LIN {X 0,Y 359.828,Z 337.187,A -85,B 0,C 180,E1 -13571.495,E2 -13571.495} C_VEL
LIN {X 0,Y 358.467,Z 346.595,A -85,B 0,C 180,E1 -13572.897,E2 -13572.897} C_VEL
LIN {X 0,Y 356.952,Z 356.826,A -85,B 0,C 180,E1 -13574.744,E2 -13574.744} C_VEL
LIN {X 0,Y 355.949,Z 365.054,A -85,B 0,C 180,E1 -13576.585,E2 -13576.585} C_VEL
LIN {X 0,Y 354.906,Z 372.31,A -85,B 0,C 180,E1 -13578.579,E2 -13578.579} C_VEL
LIN {X 0,Y 354.13,Z 378.825,A -85,B 0,C 180,E1 -13580.865,E2 -13580.865} C_VEL
LIN {X 0,Y 353.677,Z 383.707,A -85,B 0,C 180,E1 -13583.153,E2 -13583.153} C_VEL
LIN {X 0,Y 353.389,Z 387.105,A -85,B 0,C 180,E1 -13585.437,E2 -13585.437} C_VEL
LIN {X 0,Y 353.199,Z 389.123,A -85,B 0,C 180,E1 -13587.719,E2 -13587.719} C_VEL
LIN {X 0,Y 353.194,Z 389.814,A -85,B 0,C 180,E1 -13590,E2 -13590} C_VEL
LIN {X 0,Y 353.198,Z 389.189,A -85,B 0,C 180,E1 -13592.281,E2 -13592.281} C_VEL
LIN {X 0,Y 353.386,Z 387.229,A -85,B 0,C 180,E1 -13594.563,E2 -13594.563} C_VEL
LIN {X 0,Y 353.675,Z 383.892,A -85,B 0,C 180,E1 -13596.848,E2 -13596.848} C_VEL
LIN {X 0,Y 354.107,Z 379.078,A -85,B 0,C 180,E1 -13599.136,E2 -13599.136} C_VEL
LIN {X 0,Y 354.636,Z 374.431,A -85,B 0,C 180,E1 -13600.852,E2 -13600.852} C_VEL
LIN {X 0,Y 355.584,Z 367.668,A -85,B 0,C 180,E1 -13602.847,E2 -13602.847} C_VEL
LIN {X 0,Y 356.525,Z 360.612,A -85,B 0,C 180,E1 -13604.557,E2 -13604.557} C_VEL
LIN {X 0,Y 357.678,Z 352.114,A -85,B 0,C 180,E1 -13606.26,E2 -13606.26} C_VEL
LIN {X 0,Y 359.22,Z 341.807,A -85,B 0,C 180,E1 -13607.948,E2 -13607.948} C_VEL
LIN {X 0,Y 360.78,Z 330.276,A -85,B 0,C 180,E1 -13609.487,E2 -13609.487} C_VEL
LIN {X 0,Y 362.233,Z 318.754,A -85,B 0,C 180,E1 -13610.738,E2 -13610.738} C_VEL
LIN {X 0,Y 363.624,Z 305.23,A -85,B 0,C 180,E1 -13611.916,E2 -13611.916} C_VEL
LIN {X 0,Y 364.064,Z 298.662,A -85,B 0,C 180,E1 -13612.398,E2 -13612.398} C_VEL
LIN {X 0,Y 361.429,Z 285.746,A -85,B 0,C 180,E1 -13613.406,E2 -13613.406} C_VEL
LIN {X 0,Y 357.948,Z 272.835,A -85,B 0,C 180,E1 -13614.268,E2 -13614.268} C_VEL
LIN {X 0,Y 354.079,Z 260.487,A -85,B 0,C 180,E1 -13614.972,E2 -13614.972} C_VEL
LIN {X 0,Y 354.298,Z 256.381,A -85,B 0,C 180,E1 -13618.43,E2 -13618.43} C_VEL
LIN {X 0,Y 354.484,Z 253.656,A -85,B 0,C 180,E1 -13620.771,E2 -13620.771} C_VEL
LIN {X 0,Y 353.931,Z 252.674,A -85,B 0,C 180,E1 -13621.708,E2 -13621.708} C_VEL
LIN {X 0,Y 351.187,Z 251.333,A -85,B 0,C 180,E1 -13623.242,E2 -13623.242} C_VEL
LIN {X 0,Y 348.857,Z 250.304,A -85,B 0,C 180,E1 -13624.486,E2 -13624.486} C_VEL
LIN {X 0,Y 347.923,Z 249.415,A -85,B 0,C 180,E1 -13625.443,E2 -13625.443} C_VEL
LIN {X 0,Y 347.886,Z 249.081,A -85,B 0,C 180,E1 -13625.766,E2 -13625.766} C_VEL
LIN {X 0,Y 347.949,Z 246.009,A -85,B 0,C 180,E1 -13628.767,E2 -13628.767} C_VEL
LIN {X 0,Y 347.764,Z 243.044,A -85,B 0,C 180,E1 -13631.829,E2 -13631.829} C_VEL
LIN {X 0,Y 347.707,Z 242.802,A -85,B 0,C 180,E1 -13635.027,E2 -13635.027} C_VEL
LIN {X 0,Y 347.743,Z 242.796,A -85,B 0,C 180,E1 -13638.399,E2 -13638.399} C_VEL
LIN {X 0,Y 347.759,Z 242.794,A -85,B 0,C 180,E1 -13642.679,E2 -13642.679} C_VEL
LIN {X 0,Y 347.751,Z 242.795,A -85,B 0,C 180,E1 -13645.956,E2 -13645.956} C_VEL
LIN {X 0,Y 347.752,Z 242.794,A -85,B 0,C 180,E1 -13649.652,E2 -13649.652} C_VEL
LIN {X 0,Y 347.833,Z 242.783,A -85,B 0,C 180,E1 -13653.608,E2 -13653.608} C_VEL
LIN {X 0,Y 347.788,Z 242.789,A -85,B 0,C 180,E1 -13656.162,E2 -13656.162} C_VEL
LIN {X 0,Y 347.809,Z 242.783,A -85,B 0,C 180,E1 -13659.909,E2 -13659.909} C_VEL
LIN {X 0,Y 347.869,Z 242.779,A -85,B 0,C 180,E1 -13662.359,E2 -13662.359} C_VEL
LIN {X 0,Y 347.9,Z 242.773,A -85,B 0,C 180,E1 -13665.971,E2 -13665.971} C_VEL
LIN {X 0,Y 347.899,Z 242.772,A -85,B 0,C 180,E1 -13669.525,E2 -13669.525} C_VEL
LIN {X 0,Y 348.081,Z 242.751,A -85,B 0,C 180,E1 -13673.042,E2 -13673.042} C_VEL
LIN {X 0,Y 348.205,Z 242.734,A -85,B 0,C 180,E1 -13677.686,E2 -13677.686} C_VEL
LIN {X 0,Y 348.151,Z 242.743,A -85,B 0,C 180,E1 -13681.157,E2 -13681.157} C_VEL
LIN {X 0,Y 348.208,Z 242.733,A -85,B 0,C 180,E1 -13682.313,E2 -13682.313} C_VEL
LIN {X 0,Y 348.058,Z 242.753,A -85,B 0,C 180,E1 -13686.959,E2 -13686.959} C_VEL
LIN {X 0,Y 347.899,Z 242.774,A -85,B 0,C 180,E1 -13690.475,E2 -13690.475} C_VEL
LIN {X 0,Y 347.901,Z 242.775,A -85,B 0,C 180,E1 -13694.15,E2 -13694.15} C_VEL
LIN {X 0,Y 347.832,Z 242.783,A -85,B 0,C 180,E1 -13698.259,E2 -13698.259} C_VEL
LIN {X 0,Y 347.77,Z 242.791,A -85,B 0,C 180,E1 -13701.626,E2 -13701.626} C_VEL
LIN {X 0,Y 347.77,Z 242.787,A -85,B 0,C 180,E1 -13705.112,E2 -13705.112} C_VEL
LIN {X 0,Y 347.747,Z 242.795,A -85,B 0,C 180,E1 -13709.015,E2 -13709.015} C_VEL
LIN {X 0,Y 347.74,Z 242.793,A -85,B 0,C 180,E1 -13711.914,E2 -13711.914} C_VEL
LIN {X 0,Y 347.79,Z 242.793,A -85,B 0,C 180,E1 -13715.875,E2 -13715.875} C_VEL
LIN {X 0,Y 347.754,Z 242.795,A -85,B 0,C 180,E1 -13718.792,E2 -13718.792} C_VEL
LIN {X 0,Y 347.773,Z 242.876,A -85,B 0,C 180,E1 -13722.962,E2 -13722.962} C_VEL
LIN {X 0,Y 348.43,Z 246.978,A -85,B 0,C 180,E1 -13726.564,E2 -13726.564} C_VEL
LIN {X 0,Y 348.931,Z 251.04,A -85,B 0,C 180,E1 -13729.869,E2 -13729.869} C_VEL
LIN {X 0,Y 348.958,Z 253.507,A -85,B 0,C 180,E1 -13731.763,E2 -13731.763} C_VEL
LIN {X 0,Y 348.65,Z 256.872,A -85,B 0,C 180,E1 -13734.227,E2 -13734.227} C_VEL
LIN {X 0,Y 348.101,Z 262.637,A -85,B 0,C 180,E1 -13738.336,E2 -13738.336} C_VEL
LIN {X 0,Y 347.747,Z 266.494,A -85,B 0,C 180,E1 -13740.984,E2 -13740.984} C_VEL
LIN {X 0,Y 347.238,Z 271.759,A -85,B 0,C 180,E1 -13744.526,E2 -13744.526} C_VEL
LIN {X 0,Y 351.846,Z 288.484,A -85,B 0,C 180,E1 -13745.474,E2 -13745.474} C_VEL
LIN {X 0,Y 354.51,Z 300.834,A -85,B 0,C 180,E1 -13746.312,E2 -13746.312} C_VEL
LIN {X 0,Y 356.336,Z 312.535,A -85,B 0,C 180,E1 -13747.231,E2 -13747.231} C_VEL
LIN {X 0,Y 356.681,Z 316.48,A -85,B 0,C 180,E1 -13747.559,E2 -13747.559} C_VEL
LIN {X 0,Y 355.212,Z 330.023,A -85,B 0,C 180,E1 -13748.725,E2 -13748.725} C_VEL
LIN {X 0,Y 353.479,Z 342.684,A -85,B 0,C 180,E1 -13750.093,E2 -13750.093} C_VEL
LIN {X 0,Y 351.824,Z 354.335,A -85,B 0,C 180,E1 -13751.662,E2 -13751.662} C_VEL
LIN {X 0,Y 350.3,Z 364.758,A -85,B 0,C 180,E1 -13753.387,E2 -13753.387} C_VEL
LIN {X 0,Y 349.048,Z 374.137,A -85,B 0,C 180,E1 -13755.304,E2 -13755.304} C_VEL
LIN {X 0,Y 348.046,Z 381.599,A -85,B 0,C 180,E1 -13757.166,E2 -13757.166} C_VEL
LIN {X 0,Y 347.207,Z 387.367,A -85,B 0,C 180,E1 -13758.913,E2 -13758.913} C_VEL
LIN {X 0,Y 346.726,Z 392.095,A -85,B 0,C 180,E1 -13760.668,E2 -13760.668} C_VEL
LIN {X 0,Y 346.337,Z 396.996,A -85,B 0,C 180,E1 -13763.007,E2 -13763.007} C_VEL
LIN {X 0,Y 346.143,Z 400.404,A -85,B 0,C 180,E1 -13765.341,E2 -13765.341} C_VEL
LIN {X 0,Y 346.053,Z 402.419,A -85,B 0,C 180,E1 -13767.672,E2 -13767.672} C_VEL
LIN {X 0,Y 346.092,Z 403.086,A -85,B 0,C 180,E1 -13770,E2 -13770} C_VEL
LIN {X 0,Y 346.053,Z 402.413,A -85,B 0,C 180,E1 -13772.328,E2 -13772.328} C_VEL
LIN {X 0,Y 346.14,Z 400.393,A -85,B 0,C 180,E1 -13774.658,E2 -13774.658} C_VEL
LIN {X 0,Y 346.337,Z 396.976,A -85,B 0,C 180,E1 -13776.993,E2 -13776.993} C_VEL
LIN {X 0,Y 346.716,Z 392.062,A -85,B 0,C 180,E1 -13779.332,E2 -13779.332} C_VEL
LIN {X 0,Y 347.431,Z 385.508,A -85,B 0,C 180,E1 -13781.671,E2 -13781.671} C_VEL
LIN {X 0,Y 348.302,Z 379.34,A -85,B 0,C 180,E1 -13783.417,E2 -13783.417} C_VEL
LIN {X 0,Y 349.285,Z 371.939,A -85,B 0,C 180,E1 -13785.163,E2 -13785.163} C_VEL
LIN {X 0,Y 350.526,Z 363.049,A -85,B 0,C 180,E1 -13786.901,E2 -13786.901} C_VEL
LIN {X 0,Y 352.091,Z 352.286,A -85,B 0,C 180,E1 -13788.625,E2 -13788.625} C_VEL
LIN {X 0,Y 353.64,Z 341.395,A -85,B 0,C 180,E1 -13790.048,E2 -13790.048} C_VEL
LIN {X 0,Y 355.281,Z 329.679,A -85,B 0,C 180,E1 -13791.293,E2 -13791.293} C_VEL
LIN {X 0,Y 356.654,Z 316.345,A -85,B 0,C 180,E1 -13792.439,E2 -13792.439} C_VEL
LIN {X 0,Y 355.141,Z 304.648,A -85,B 0,C 180,E1 -13793.392,E2 -13793.392} C_VEL
LIN {X 0,Y 352.32,Z 290.353,A -85,B 0,C 180,E1 -13794.393,E2 -13794.393} C_VEL
LIN {X 0,Y 348.517,Z 276.599,A -85,B 0,C 180,E1 -13795.205,E2 -13795.205} C_VEL
LIN {X 0,Y 347.245,Z 271.771,A -85,B 0,C 180,E1 -13795.448,E2 -13795.448} C_VEL
LIN {X 0,Y 347.745,Z 266.467,A -85,B 0,C 180,E1 -13799.015,E2 -13799.015} C_VEL
LIN {X 0,Y 348.262,Z 260.693,A -85,B 0,C 180,E1 -13803.016,E2 -13803.016} C_VEL
LIN {X 0,Y 348.722,Z 256.134,A -85,B 0,C 180,E1 -13806.279,E2 -13806.279} C_VEL
LIN {X 0,Y 348.962,Z 252.942,A -85,B 0,C 180,E1 -13808.633,E2 -13808.633} C_VEL
LIN {X 0,Y 348.927,Z 250.987,A -85,B 0,C 180,E1 -13810.131,E2 -13810.131} C_VEL
LIN {X 0,Y 348.416,Z 246.945,A -85,B 0,C 180,E1 -13813.434,E2 -13813.434} C_VEL
LIN {X 0,Y 347.845,Z 243.239,A -85,B 0,C 180,E1 -13816.666,E2 -13816.666} C_VEL
LIN {X 0,Y 347.755,Z 242.797,A -85,B 0,C 180,E1 -13817.226,E2 -13817.226} C_VEL
LIN {X 0,Y 347.752,Z 242.796,A -85,B 0,C 180,E1 -13821.207,E2 -13821.207} C_VEL
LIN {X 0,Y 347.789,Z 242.792,A -85,B 0,C 180,E1 -13824.125,E2 -13824.125} C_VEL
LIN {X 0,Y 347.739,Z 242.796,A -85,B 0,C 180,E1 -13828.086,E2 -13828.086} C_VEL
LIN {X 0,Y 347.747,Z 242.795,A -85,B 0,C 180,E1 -13830.985,E2 -13830.985} C_VEL
LIN {X 0,Y 347.751,Z 242.793,A -85,B 0,C 180,E1 -13833.601,E2 -13833.601} C_VEL
LIN {X 0,Y 347.77,Z 242.791,A -85,B 0,C 180,E1 -13836.161,E2 -13836.161} C_VEL
LIN {X 0,Y 347.807,Z 242.786,A -85,B 0,C 180,E1 -13839.909,E2 -13839.909} C_VEL
LIN {X 0,Y 347.834,Z 242.783,A -85,B 0,C 180,E1 -13843.568,E2 -13843.568} C_VEL
LIN {X 0,Y 347.891,Z 242.777,A -85,B 0,C 180,E1 -13847.161,E2 -13847.161} C_VEL
LIN {X 0,Y 347.936,Z 242.77,A -85,B 0,C 180,E1 -13850.701,E2 -13850.701} C_VEL
LIN {X 0,Y 348.045,Z 242.755,A -85,B 0,C 180,E1 -13854.205,E2 -13854.205} C_VEL
LIN {X 0,Y 348.207,Z 242.735,A -85,B 0,C 180,E1 -13857.687,E2 -13857.687} C_VEL
LIN {X 0,Y 348.284,Z 242.728,A -85,B 0,C 180,E1 -13860,E2 -13860} C_VEL
LIN {X 0,Y 348.203,Z 242.735,A -85,B 0,C 180,E1 -13862.314,E2 -13862.314} C_VEL
LIN {X 0,Y 348.092,Z 242.75,A -85,B 0,C 180,E1 -13866.958,E2 -13866.958} C_VEL
LIN {X 0,Y 347.93,Z 242.77,A -85,B 0,C 180,E1 -13870.474,E2 -13870.474} C_VEL
LIN {X 0,Y 347.9,Z 242.773,A -85,B 0,C 180,E1 -13874.15,E2 -13874.15} C_VEL
LIN {X 0,Y 347.893,Z 242.775,A -85,B 0,C 180,E1 -13878.291,E2 -13878.291} C_VEL
LIN {X 0,Y 347.769,Z 242.789,A -85,B 0,C 180,E1 -13881.626,E2 -13881.626} C_VEL
LIN {X 0,Y 347.813,Z 242.784,A -85,B 0,C 180,E1 -13885.109,E2 -13885.109} C_VEL
LIN {X 0,Y 347.81,Z 242.786,A -85,B 0,C 180,E1 -13887.694,E2 -13887.694} C_VEL
LIN {X 0,Y 347.751,Z 242.793,A -85,B 0,C 180,E1 -13890.348,E2 -13890.348} C_VEL
LIN {X 0,Y 347.749,Z 242.794,A -85,B 0,C 180,E1 -13894.044,E2 -13894.044} C_VEL
LIN {X 0,Y 347.758,Z 242.794,A -85,B 0,C 180,E1 -13897.322,E2 -13897.322} C_VEL
LIN {X 0,Y 347.742,Z 242.796,A -85,B 0,C 180,E1 -13901.601,E2 -13901.601} C_VEL
LIN {X 0,Y 347.706,Z 242.8,A -85,B 0,C 180,E1 -13905.027,E2 -13905.027} C_VEL
LIN {X 0,Y 347.763,Z 242.921,A -85,B 0,C 180,E1 -13908.172,E2 -13908.172} C_VEL
LIN {X 0,Y 347.964,Z 245.902,A -85,B 0,C 180,E1 -13911.235,E2 -13911.235} C_VEL
LIN {X 0,Y 347.897,Z 248.859,A -85,B 0,C 180,E1 -13914.138,E2 -13914.138} C_VEL
LIN {X 0,Y 347.633,Z 251.861,A -85,B 0,C 180,E1 -13916.917,E2 -13916.917} C_VEL
LIN {X 0,Y 347.313,Z 255.844,A -85,B 0,C 180,E1 -13920.473,E2 -13920.473} C_VEL
LIN {X 0,Y 347.05,Z 260.626,A -85,B 0,C 180,E1 -13924.592,E2 -13924.592} C_VEL
LIN {X 0,Y 352.324,Z 277.531,A -85,B 0,C 180,E1 -13925.624,E2 -13925.624} C_VEL
LIN {X 0,Y 355.52,Z 290.249,A -85,B 0,C 180,E1 -13926.55,E2 -13926.55} C_VEL
LIN {X 0,Y 357.453,Z 300.982,A -85,B 0,C 180,E1 -13927.439,E2 -13927.439} C_VEL
LIN {X 0,Y 356.211,Z 313.402,A -85,B 0,C 180,E1 -13928.44,E2 -13928.44} C_VEL
LIN {X 0,Y 354.679,Z 325.974,A -85,B 0,C 180,E1 -13929.71,E2 -13929.71} C_VEL
LIN {X 0,Y 353.104,Z 337.325,A -85,B 0,C 180,E1 -13931.129,E2 -13931.129} C_VEL
LIN {X 0,Y 351.68,Z 346.733,A -85,B 0,C 180,E1 -13932.557,E2 -13932.557} C_VEL
LIN {X 0,Y 350.18,Z 356.452,A -85,B 0,C 180,E1 -13934.334,E2 -13934.334} C_VEL
LIN {X 0,Y 349.021,Z 365.191,A -85,B 0,C 180,E1 -13936.314,E2 -13936.314} C_VEL
LIN {X 0,Y 347.905,Z 372.448,A -85,B 0,C 180,E1 -13938.346,E2 -13938.346} C_VEL
LIN {X 0,Y 347.111,Z 378.961,A -85,B 0,C 180,E1 -13940.678,E2 -13940.678} C_VEL
LIN {X 0,Y 346.613,Z 383.843,A -85,B 0,C 180,E1 -13943.012,E2 -13943.012} C_VEL
LIN {X 0,Y 346.308,Z 387.24,A -85,B 0,C 180,E1 -13945.344,E2 -13945.344} C_VEL
LIN {X 0,Y 346.11,Z 389.258,A -85,B 0,C 180,E1 -13947.673,E2 -13947.673} C_VEL
LIN {X 0,Y 346.095,Z 389.949,A -85,B 0,C 180,E1 -13950,E2 -13950} C_VEL
LIN {X 0,Y 346.109,Z 389.323,A -85,B 0,C 180,E1 -13952.328,E2 -13952.328} C_VEL
LIN {X 0,Y 346.304,Z 387.363,A -85,B 0,C 180,E1 -13954.656,E2 -13954.656} C_VEL
LIN {X 0,Y 346.612,Z 384.026,A -85,B 0,C 180,E1 -13956.988,E2 -13956.988} C_VEL
LIN {X 0,Y 347.093,Z 379.212,A -85,B 0,C 180,E1 -13959.322,E2 -13959.322} C_VEL
LIN {X 0,Y 347.844,Z 372.765,A -85,B 0,C 180,E1 -13961.657,E2 -13961.657} C_VEL
LIN {X 0,Y 348.99,Z 365.579,A -85,B 0,C 180,E1 -13963.687,E2 -13963.687} C_VEL
LIN {X 0,Y 350.126,Z 356.973,A -85,B 0,C 180,E1 -13965.663,E2 -13965.663} C_VEL
LIN {X 0,Y 351.645,Z 347.35,A -85,B 0,C 180,E1 -13967.445,E2 -13967.445} C_VEL
LIN {X 0,Y 353.161,Z 337.001,A -85,B 0,C 180,E1 -13969.018,E2 -13969.018} C_VEL
LIN {X 0,Y 354.73,Z 325.578,A -85,B 0,C 180,E1 -13970.438,E2 -13970.438} C_VEL
LIN {X 0,Y 356.287,Z 312.912,A -85,B 0,C 180,E1 -13971.707,E2 -13971.707} C_VEL
LIN {X 0,Y 357.481,Z 300.595,A -85,B 0,C 180,E1 -13972.695,E2 -13972.695} C_VEL
LIN {X 0,Y 354.933,Z 287.672,A -85,B 0,C 180,E1 -13973.753,E2 -13973.753} C_VEL
LIN {X 0,Y 351.396,Z 274.214,A -85,B 0,C 180,E1 -13974.696,E2 -13974.696} C_VEL
LIN {X 0,Y 347.12,Z 261.12,A -85,B 0,C 180,E1 -13975.472,E2 -13975.472} C_VEL
LIN {X 0,Y 347.057,Z 260.623,A -85,B 0,C 180,E1 -13975.52,E2 -13975.52} C_VEL
LIN {X 0,Y 347.342,Z 255.956,A -85,B 0,C 180,E1 -13979.536,E2 -13979.536} C_VEL
LIN {X 0,Y 347.634,Z 251.985,A -85,B 0,C 180,E1 -13983.083,E2 -13983.083} C_VEL
LIN {X 0,Y 347.886,Z 249.081,A -85,B 0,C 180,E1 -13985.766,E2 -13985.766} C_VEL
LIN {X 0,Y 347.327,Z 248.172,A -85,B 0,C 180,E1 -13986.72,E2 -13986.72} C_VEL
LIN {X 0,Y 344.517,Z 247.005,A -85,B 0,C 180,E1 -13988.281,E2 -13988.281} C_VEL
LIN {X 0,Y 342.041,Z 246.131,A -85,B 0,C 180,E1 -13989.546,E2 -13989.546} C_VEL
LIN {X 0,Y 340.928,Z 245.355,A -85,B 0,C 180,E1 -13990.523,E2 -13990.523} C_VEL
LIN {X 0,Y 340.815,Z 245.056,A -85,B 0,C 180,E1 -13990.853,E2 -13990.853} C_VEL
LIN {X 0,Y 340.727,Z 243.941,A -85,B 0,C 180,E1 -13992.05,E2 -13992.05} C_VEL
LIN {X 0,Y 340.643,Z 243.682,A -85,B 0,C 180,E1 -13994.546,E2 -13994.546} C_VEL
LIN {X 0,Y 340.695,Z 243.674,A -85,B 0,C 180,E1 -13997.956,E2 -13997.956} C_VEL
LIN {X 0,Y 340.721,Z 243.668,A -85,B 0,C 180,E1 -14001.771,E2 -14001.771} C_VEL
LIN {X 0,Y 340.725,Z 243.668,A -85,B 0,C 180,E1 -14005.595,E2 -14005.595} C_VEL
LIN {X 0,Y 340.7,Z 243.672,A -85,B 0,C 180,E1 -14008.955,E2 -14008.955} C_VEL
LIN {X 0,Y 340.806,Z 243.658,A -85,B 0,C 180,E1 -14013.02,E2 -14013.02} C_VEL
LIN {X 0,Y 340.757,Z 243.661,A -85,B 0,C 180,E1 -14015.638,E2 -14015.638} C_VEL
LIN {X 0,Y 340.737,Z 243.665,A -85,B 0,C 180,E1 -14019.473,E2 -14019.473} C_VEL
LIN {X 0,Y 340.861,Z 243.652,A -85,B 0,C 180,E1 -14021.984,E2 -14021.984} C_VEL
LIN {X 0,Y 340.872,Z 243.65,A -85,B 0,C 180,E1 -14025.705,E2 -14025.705} C_VEL
LIN {X 0,Y 340.851,Z 243.65,A -85,B 0,C 180,E1 -14029.305,E2 -14029.305} C_VEL
LIN {X 0,Y 341.048,Z 243.627,A -85,B 0,C 180,E1 -14032.898,E2 -14032.898} C_VEL
LIN {X 0,Y 341.167,Z 243.611,A -85,B 0,C 180,E1 -14037.639,E2 -14037.639} C_VEL
LIN {X 0,Y 341.12,Z 243.619,A -85,B 0,C 180,E1 -14041.18,E2 -14041.18} C_VEL
LIN {X 0,Y 341.17,Z 243.61,A -85,B 0,C 180,E1 -14042.361,E2 -14042.361} C_VEL
LIN {X 0,Y 341.005,Z 243.631,A -85,B 0,C 180,E1 -14047.103,E2 -14047.103} C_VEL
LIN {X 0,Y 340.85,Z 243.652,A -85,B 0,C 180,E1 -14050.694,E2 -14050.694} C_VEL
LIN {X 0,Y 340.866,Z 243.652,A -85,B 0,C 180,E1 -14054.325,E2 -14054.325} C_VEL
LIN {X 0,Y 340.789,Z 243.66,A -85,B 0,C 180,E1 -14058.441,E2 -14058.441} C_VEL
LIN {X 0,Y 340.72,Z 243.669,A -85,B 0,C 180,E1 -14061.841,E2 -14061.841} C_VEL
LIN {X 0,Y 340.721,Z 243.664,A -85,B 0,C 180,E1 -14065.668,E2 -14065.668} C_VEL
LIN {X 0,Y 340.709,Z 243.671,A -85,B 0,C 180,E1 -14069.674,E2 -14069.674} C_VEL
LIN {X 0,Y 340.688,Z 243.675,A -85,B 0,C 180,E1 -14072.436,E2 -14072.436} C_VEL
LIN {X 0,Y 340.72,Z 243.672,A -85,B 0,C 180,E1 -14075.279,E2 -14075.279} C_VEL
LIN {X 0,Y 340.711,Z 243.673,A -85,B 0,C 180,E1 -14078.386,E2 -14078.386} C_VEL
LIN {X 0,Y 340.716,Z 243.722,A -85,B 0,C 180,E1 -14082.54,E2 -14082.54} C_VEL
LIN {X 0,Y 341.357,Z 247.68,A -85,B 0,C 180,E1 -14086.104,E2 -14086.104} C_VEL
LIN {X 0,Y 341.882,Z 251.744,A -85,B 0,C 180,E1 -14089.517,E2 -14089.517} C_VEL
LIN {X 0,Y 341.924,Z 254.813,A -85,B 0,C 180,E1 -14091.929,E2 -14091.929} C_VEL
LIN {X 0,Y 341.424,Z 259.506,A -85,B 0,C 180,E1 -14095.424,E2 -14095.424} C_VEL
LIN {X 0,Y 340.944,Z 264.434,A -85,B 0,C 180,E1 -14098.98,E2 -14098.98} C_VEL
LIN {X 0,Y 340.564,Z 268.275,A -85,B 0,C 180,E1 -14101.664,E2 -14101.664} C_VEL
LIN {X 0,Y 340.268,Z 271.798,A -85,B 0,C 180,E1 -14103.994,E2 -14103.994} C_VEL
LIN {X 0,Y 344.24,Z 285.702,A -85,B 0,C 180,E1 -14104.779,E2 -14104.779} C_VEL
LIN {X 0,Y 347.179,Z 298.328,A -85,B 0,C 180,E1 -14105.636,E2 -14105.636} C_VEL
LIN {X 0,Y 349.36,Z 311.042,A -85,B 0,C 180,E1 -14106.643,E2 -14106.643} C_VEL
LIN {X 0,Y 349.925,Z 318.302,A -85,B 0,C 180,E1 -14107.273,E2 -14107.273} C_VEL
LIN {X 0,Y 348.524,Z 330.344,A -85,B 0,C 180,E1 -14108.345,E2 -14108.345} C_VEL
LIN {X 0,Y 346.808,Z 342.553,A -85,B 0,C 180,E1 -14109.694,E2 -14109.694} C_VEL
LIN {X 0,Y 345.336,Z 352.247,A -85,B 0,C 180,E1 -14110.997,E2 -14110.997} C_VEL
LIN {X 0,Y 343.71,Z 362.992,A -85,B 0,C 180,E1 -14112.753,E2 -14112.753} C_VEL
LIN {X 0,Y 342.398,Z 371.868,A -85,B 0,C 180,E1 -14114.524,E2 -14114.524} C_VEL
LIN {X 0,Y 341.232,Z 380.377,A -85,B 0,C 180,E1 -14116.602,E2 -14116.602} C_VEL
LIN {X 0,Y 340.2,Z 387.233,A -85,B 0,C 180,E1 -14118.682,E2 -14118.682} C_VEL
LIN {X 0,Y 339.687,Z 391.961,A -85,B 0,C 180,E1 -14120.473,E2 -14120.473} C_VEL
LIN {X 0,Y 339.26,Z 396.862,A -85,B 0,C 180,E1 -14122.86,E2 -14122.86} C_VEL
LIN {X 0,Y 339.047,Z 400.27,A -85,B 0,C 180,E1 -14125.244,E2 -14125.244} C_VEL
LIN {X 0,Y 338.969,Z 402.285,A -85,B 0,C 180,E1 -14127.623,E2 -14127.623} C_VEL
LIN {X 0,Y 338.994,Z 402.951,A -85,B 0,C 180,E1 -14130,E2 -14130} C_VEL
LIN {X 0,Y 338.969,Z 402.278,A -85,B 0,C 180,E1 -14132.376,E2 -14132.376} C_VEL
LIN {X 0,Y 339.045,Z 400.257,A -85,B 0,C 180,E1 -14134.756,E2 -14134.756} C_VEL
LIN {X 0,Y 339.26,Z 396.84,A -85,B 0,C 180,E1 -14137.14,E2 -14137.14} C_VEL
LIN {X 0,Y 339.68,Z 391.926,A -85,B 0,C 180,E1 -14139.527,E2 -14139.527} C_VEL
LIN {X 0,Y 340.455,Z 385.371,A -85,B 0,C 180,E1 -14141.913,E2 -14141.913} C_VEL
LIN {X 0,Y 341.484,Z 378.081,A -85,B 0,C 180,E1 -14143.994,E2 -14143.994} C_VEL
LIN {X 0,Y 342.56,Z 370.441,A -85,B 0,C 180,E1 -14145.774,E2 -14145.774} C_VEL
LIN {X 0,Y 343.957,Z 361.279,A -85,B 0,C 180,E1 -14147.541,E2 -14147.541} C_VEL
LIN {X 0,Y 345.607,Z 350.169,A -85,B 0,C 180,E1 -14149.296,E2 -14149.296} C_VEL
LIN {X 0,Y 347.36,Z 338.831,A -85,B 0,C 180,E1 -14150.736,E2 -14150.736} C_VEL
LIN {X 0,Y 348.942,Z 327.034,A -85,B 0,C 180,E1 -14151.959,E2 -14151.959} C_VEL
LIN {X 0,Y 349.918,Z 316.488,A -85,B 0,C 180,E1 -14152.87,E2 -14152.87} C_VEL
LIN {X 0,Y 348.294,Z 304.5,A -85,B 0,C 180,E1 -14153.88,E2 -14153.88} C_VEL
LIN {X 0,Y 345.498,Z 290.644,A -85,B 0,C 180,E1 -14154.885,E2 -14154.885} C_VEL
LIN {X 0,Y 341.361,Z 275.824,A -85,B 0,C 180,E1 -14155.789,E2 -14155.789} C_VEL
LIN {X 0,Y 340.257,Z 271.653,A -85,B 0,C 180,E1 -14156.007,E2 -14156.007} C_VEL
LIN {X 0,Y 340.837,Z 265.842,A -85,B 0,C 180,E1 -14159.999,E2 -14159.999} C_VEL
LIN {X 0,Y 341.315,Z 260.561,A -85,B 0,C 180,E1 -14163.777,E2 -14163.777} C_VEL
LIN {X 0,Y 341.746,Z 256.635,A -85,B 0,C 180,E1 -14166.675,E2 -14166.675} C_VEL
LIN {X 0,Y 341.929,Z 252.828,A -85,B 0,C 180,E1 -14169.581,E2 -14169.581} C_VEL
LIN {X 0,Y 341.505,Z 248.944,A -85,B 0,C 180,E1 -14172.775,E2 -14172.775} C_VEL
LIN {X 0,Y 340.927,Z 245.069,A -85,B 0,C 180,E1 -14176.179,E2 -14176.179} C_VEL
LIN {X 0,Y 340.725,Z 243.67,A -85,B 0,C 180,E1 -14177.58,E2 -14177.58} C_VEL
LIN {X 0,Y 340.733,Z 243.67,A -85,B 0,C 180,E1 -14181.773,E2 -14181.773} C_VEL
LIN {X 0,Y 340.723,Z 243.672,A -85,B 0,C 180,E1 -14185.595,E2 -14185.595} C_VEL
LIN {X 0,Y 340.695,Z 243.674,A -85,B 0,C 180,E1 -14188.955,E2 -14188.955} C_VEL
LIN {X 0,Y 340.721,Z 243.668,A -85,B 0,C 180,E1 -14193.013,E2 -14193.013} C_VEL
LIN {X 0,Y 340.742,Z 243.668,A -85,B 0,C 180,E1 -14195.637,E2 -14195.637} C_VEL
LIN {X 0,Y 340.735,Z 243.667,A -85,B 0,C 180,E1 -14199.473,E2 -14199.473} C_VEL
LIN {X 0,Y 340.794,Z 243.658,A -85,B 0,C 180,E1 -14201.981,E2 -14201.981} C_VEL
LIN {X 0,Y 340.871,Z 243.647,A -85,B 0,C 180,E1 -14205.705,E2 -14205.705} C_VEL
LIN {X 0,Y 340.849,Z 243.646,A -85,B 0,C 180,E1 -14209.306,E2 -14209.306} C_VEL
LIN {X 0,Y 341.004,Z 243.632,A -85,B 0,C 180,E1 -14212.897,E2 -14212.897} C_VEL
LIN {X 0,Y 341.169,Z 243.612,A -85,B 0,C 180,E1 -14217.639,E2 -14217.639} C_VEL
LIN {X 0,Y 341.236,Z 243.606,A -85,B 0,C 180,E1 -14220,E2 -14220} C_VEL
LIN {X 0,Y 341.165,Z 243.612,A -85,B 0,C 180,E1 -14222.361,E2 -14222.361} C_VEL
LIN {X 0,Y 341.06,Z 243.625,A -85,B 0,C 180,E1 -14227.102,E2 -14227.102} C_VEL
LIN {X 0,Y 340.873,Z 243.649,A -85,B 0,C 180,E1 -14230.694,E2 -14230.694} C_VEL
LIN {X 0,Y 340.865,Z 243.65,A -85,B 0,C 180,E1 -14234.325,E2 -14234.325} C_VEL
LIN {X 0,Y 340.84,Z 243.653,A -85,B 0,C 180,E1 -14238.467,E2 -14238.467} C_VEL
LIN {X 0,Y 340.719,Z 243.667,A -85,B 0,C 180,E1 -14241.842,E2 -14241.842} C_VEL
LIN {X 0,Y 340.773,Z 243.663,A -85,B 0,C 180,E1 -14245.664,E2 -14245.664} C_VEL
LIN {X 0,Y 340.73,Z 243.666,A -85,B 0,C 180,E1 -14248.321,E2 -14248.321} C_VEL
LIN {X 0,Y 340.699,Z 243.672,A -85,B 0,C 180,E1 -14251.045,E2 -14251.045} C_VEL
LIN {X 0,Y 340.719,Z 243.67,A -85,B 0,C 180,E1 -14255.279,E2 -14255.279} C_VEL
LIN {X 0,Y 340.695,Z 243.672,A -85,B 0,C 180,E1 -14258.383,E2 -14258.383} C_VEL
LIN {X 0,Y 340.694,Z 243.674,A -85,B 0,C 180,E1 -14262.044,E2 -14262.044} C_VEL
LIN {X 0,Y 340.653,Z 243.679,A -85,B 0,C 180,E1 -14266.227,E2 -14266.227} C_VEL
LIN {X 0,Y 340.726,Z 243.821,A -85,B 0,C 180,E1 -14267.95,E2 -14267.95} C_VEL
LIN {X 0,Y 340.943,Z 246.007,A -85,B 0,C 180,E1 -14270.282,E2 -14270.282} C_VEL
LIN {X 0,Y 340.882,Z 249.225,A -85,B 0,C 180,E1 -14273.52,E2 -14273.52} C_VEL
LIN {X 0,Y 340.673,Z 251.992,A -85,B 0,C 180,E1 -14276.151,E2 -14276.151} C_VEL
LIN {X 0,Y 340.39,Z 255.003,A -85,B 0,C 180,E1 -14278.924,E2 -14278.924} C_VEL
LIN {X 0,Y 340.106,Z 259.528,A -85,B 0,C 180,E1 -14282.96,E2 -14282.96} C_VEL
LIN {X 0,Y 340.031,Z 260.777,A -85,B 0,C 180,E1 -14284.052,E2 -14284.052} C_VEL
LIN {X 0,Y 341.739,Z 266.22,A -85,B 0,C 180,E1 -14284.352,E2 -14284.352} C_VEL
LIN {X 0,Y 345.913,Z 279.449,A -85,B 0,C 180,E1 -14285.229,E2 -14285.229} C_VEL
LIN {X 0,Y 349.175,Z 292.874,A -85,B 0,C 180,E1 -14286.262,E2 -14286.262} C_VEL
LIN {X 0,Y 350.782,Z 302.012,A -85,B 0,C 180,E1 -14287.056,E2 -14287.056} C_VEL
LIN {X 0,Y 349.439,Z 315.12,A -85,B 0,C 180,E1 -14288.156,E2 -14288.156} C_VEL
LIN {X 0,Y 347.857,Z 327.385,A -85,B 0,C 180,E1 -14289.449,E2 -14289.449} C_VEL
LIN {X 0,Y 346.385,Z 337.464,A -85,B 0,C 180,E1 -14290.749,E2 -14290.749} C_VEL
LIN {X 0,Y 344.892,Z 346.872,A -85,B 0,C 180,E1 -14292.202,E2 -14292.202} C_VEL
LIN {X 0,Y 343.387,Z 356.324,A -85,B 0,C 180,E1 -14293.961,E2 -14293.961} C_VEL
LIN {X 0,Y 342.11,Z 365.328,A -85,B 0,C 180,E1 -14296.032,E2 -14296.032} C_VEL
LIN {X 0,Y 340.916,Z 372.585,A -85,B 0,C 180,E1 -14298.103,E2 -14298.103} C_VEL
LIN {X 0,Y 340.069,Z 379.097,A -85,B 0,C 180,E1 -14300.484,E2 -14300.484} C_VEL
LIN {X 0,Y 339.55,Z 383.979,A -85,B 0,C 180,E1 -14302.866,E2 -14302.866} C_VEL
LIN {X 0,Y 339.229,Z 387.375,A -85,B 0,C 180,E1 -14305.247,E2 -14305.247} C_VEL
LIN {X 0,Y 339.024,Z 389.393,A -85,B 0,C 180,E1 -14307.624,E2 -14307.624} C_VEL
LIN {X 0,Y 338.998,Z 390.084,A -85,B 0,C 180,E1 -14310,E2 -14310} C_VEL
LIN {X 0,Y 339.023,Z 389.457,A -85,B 0,C 180,E1 -14312.376,E2 -14312.376} C_VEL
LIN {X 0,Y 339.226,Z 387.497,A -85,B 0,C 180,E1 -14314.754,E2 -14314.754} C_VEL
LIN {X 0,Y 339.549,Z 384.16,A -85,B 0,C 180,E1 -14317.134,E2 -14317.134} C_VEL
LIN {X 0,Y 340.051,Z 379.346,A -85,B 0,C 180,E1 -14319.517,E2 -14319.517} C_VEL
LIN {X 0,Y 340.857,Z 372.898,A -85,B 0,C 180,E1 -14321.899,E2 -14321.899} C_VEL
LIN {X 0,Y 342.086,Z 365.712,A -85,B 0,C 180,E1 -14323.969,E2 -14323.969} C_VEL
LIN {X 0,Y 343.272,Z 357.106,A -85,B 0,C 180,E1 -14325.984,E2 -14325.984} C_VEL
LIN {X 0,Y 344.852,Z 347.483,A -85,B 0,C 180,E1 -14327.8,E2 -14327.8} C_VEL
LIN {X 0,Y 346.429,Z 337.133,A -85,B 0,C 180,E1 -14329.403,E2 -14329.403} C_VEL
LIN {X 0,Y 348.087,Z 325.708,A -85,B 0,C 180,E1 -14330.846,E2 -14330.846} C_VEL
LIN {X 0,Y 349.691,Z 313.094,A -85,B 0,C 180,E1 -14332.133,E2 -14332.133} C_VEL
LIN {X 0,Y 350.76,Z 301.487,A -85,B 0,C 180,E1 -14333.095,E2 -14333.095} C_VEL
LIN {X 0,Y 348.256,Z 288.795,A -85,B 0,C 180,E1 -14334.177,E2 -14334.177} C_VEL
LIN {X 0,Y 344.843,Z 275.803,A -85,B 0,C 180,E1 -14335.133,E2 -14335.133} C_VEL
LIN {X 0,Y 340.087,Z 261.198,A -85,B 0,C 180,E1 -14336.039,E2 -14336.039} C_VEL
LIN {X 0,Y 340.052,Z 260.737,A -85,B 0,C 180,E1 -14336.093,E2 -14336.093} C_VEL
LIN {X 0,Y 340.309,Z 256.497,A -85,B 0,C 180,E1 -14339.844,E2 -14339.844} C_VEL
LIN {X 0,Y 340.677,Z 252.115,A -85,B 0,C 180,E1 -14343.849,E2 -14343.849} C_VEL
LIN {X 0,Y 340.885,Z 249.101,A -85,B 0,C 180,E1 -14346.719,E2 -14346.719} C_VEL
LIN {X 0,Y 340.926,Z 246.128,A -85,B 0,C 180,E1 -14349.721,E2 -14349.721} C_VEL
LIN {X 0,Y 340.815,Z 245.056,A -85,B 0,C 180,E1 -14350.853,E2 -14350.853} C_VEL
LIN {X 0,Y 340.077,Z 244.403,A -85,B 0,C 180,E1 -14351.832,E2 -14351.832} C_VEL
LIN {X 0,Y 337.174,Z 244.194,A -85,B 0,C 180,E1 -14353.435,E2 -14353.435} C_VEL
LIN {X 0,Y 334.741,Z 244.418,A -85,B 0,C 180,E1 -14354.737,E2 -14354.737} C_VEL
LIN {X 0,Y 333.686,Z 244.55,A -85,B 0,C 180,E1 -14355.746,E2 -14355.746} C_VEL
LIN {X 0,Y 333.591,Z 244.56,A -85,B 0,C 180,E1 -14356.087,E2 -14356.087} C_VEL
LIN {X 0,Y 333.604,Z 244.557,A -85,B 0,C 180,E1 -14359.324,E2 -14359.324} C_VEL
LIN {X 0,Y 333.665,Z 244.549,A -85,B 0,C 180,E1 -14363.168,E2 -14363.168} C_VEL
LIN {X 0,Y 333.676,Z 244.546,A -85,B 0,C 180,E1 -14365.341,E2 -14365.341} C_VEL
LIN {X 0,Y 333.693,Z 244.545,A -85,B 0,C 180,E1 -14369.637,E2 -14369.637} C_VEL
LIN {X 0,Y 333.742,Z 244.539,A -85,B 0,C 180,E1 -14372.401,E2 -14372.401} C_VEL
LIN {X 0,Y 333.728,Z 244.534,A -85,B 0,C 180,E1 -14375.091,E2 -14375.091} C_VEL
LIN {X 0,Y 333.676,Z 244.548,A -85,B 0,C 180,E1 -14379.019,E2 -14379.019} C_VEL
LIN {X 0,Y 333.796,Z 244.53,A -85,B 0,C 180,E1 -14381.589,E2 -14381.589} C_VEL
LIN {X 0,Y 333.811,Z 244.531,A -85,B 0,C 180,E1 -14385.576,E2 -14385.576} C_VEL
LIN {X 0,Y 333.82,Z 244.527,A -85,B 0,C 180,E1 -14389.077,E2 -14389.077} C_VEL
LIN {X 0,Y 333.995,Z 244.505,A -85,B 0,C 180,E1 -14392.747,E2 -14392.747} C_VEL
LIN {X 0,Y 333.802,Z 244.531,A -85,B 0,C 180,E1 -14395.169,E2 -14395.169} C_VEL
LIN {X 0,Y 334.104,Z 244.491,A -85,B 0,C 180,E1 -14397.589,E2 -14397.589} C_VEL
LIN {X 0,Y 334.088,Z 244.495,A -85,B 0,C 180,E1 -14401.205,E2 -14401.205} C_VEL
LIN {X 0,Y 334.107,Z 244.489,A -85,B 0,C 180,E1 -14402.411,E2 -14402.411} C_VEL
LIN {X 0,Y 333.994,Z 244.506,A -85,B 0,C 180,E1 -14406.039,E2 -14406.039} C_VEL
LIN {X 0,Y 333.823,Z 244.529,A -85,B 0,C 180,E1 -14409.696,E2 -14409.696} C_VEL
LIN {X 0,Y 333.799,Z 244.532,A -85,B 0,C 180,E1 -14413.391,E2 -14413.391} C_VEL
LIN {X 0,Y 333.721,Z 244.54,A -85,B 0,C 180,E1 -14417.147,E2 -14417.147} C_VEL
LIN {X 0,Y 333.719,Z 244.543,A -85,B 0,C 180,E1 -14419.691,E2 -14419.691} C_VEL
LIN {X 0,Y 333.661,Z 244.547,A -85,B 0,C 180,E1 -14423.591,E2 -14423.591} C_VEL
LIN {X 0,Y 333.657,Z 244.545,A -85,B 0,C 180,E1 -14426.253,E2 -14426.253} C_VEL
LIN {X 0,Y 333.659,Z 244.549,A -85,B 0,C 180,E1 -14430.366,E2 -14430.366} C_VEL
LIN {X 0,Y 333.638,Z 244.55,A -85,B 0,C 180,E1 -14433.208,E2 -14433.208} C_VEL
LIN {X 0,Y 333.678,Z 244.551,A -85,B 0,C 180,E1 -14436.139,E2 -14436.139} C_VEL
LIN {X 0,Y 333.648,Z 244.552,A -85,B 0,C 180,E1 -14439.192,E2 -14439.192} C_VEL
LIN {X 0,Y 333.71,Z 244.635,A -85,B 0,C 180,E1 -14442.167,E2 -14442.167} C_VEL
LIN {X 0,Y 334.378,Z 248.879,A -85,B 0,C 180,E1 -14446.084,E2 -14446.084} C_VEL
LIN {X 0,Y 334.874,Z 252.747,A -85,B 0,C 180,E1 -14449.413,E2 -14449.413} C_VEL
LIN {X 0,Y 334.932,Z 254.695,A -85,B 0,C 180,E1 -14450.986,E2 -14450.986} C_VEL
LIN {X 0,Y 334.591,Z 258.561,A -85,B 0,C 180,E1 -14453.975,E2 -14453.975} C_VEL
LIN {X 0,Y 334.142,Z 262.957,A -85,B 0,C 180,E1 -14457.28,E2 -14457.28} C_VEL
LIN {X 0,Y 333.838,Z 266.252,A -85,B 0,C 180,E1 -14459.671,E2 -14459.671} C_VEL
LIN {X 0,Y 333.295,Z 271.525,A -85,B 0,C 180,E1 -14463.402,E2 -14463.402} C_VEL
LIN {X 0,Y 334.978,Z 277.433,A -85,B 0,C 180,E1 -14463.716,E2 -14463.716} C_VEL
LIN {X 0,Y 338.849,Z 291.762,A -85,B 0,C 180,E1 -14464.64,E2 -14464.64} C_VEL
LIN {X 0,Y 341.444,Z 304.438,A -85,B 0,C 180,E1 -14465.597,E2 -14465.597} C_VEL
LIN {X 0,Y 343.223,Z 316.766,A -85,B 0,C 180,E1 -14466.677,E2 -14466.677} C_VEL
LIN {X 0,Y 342.789,Z 323.438,A -85,B 0,C 180,E1 -14467.261,E2 -14467.261} C_VEL
LIN {X 0,Y 341.245,Z 334.949,A -85,B 0,C 180,E1 -14468.399,E2 -14468.399} C_VEL
LIN {X 0,Y 339.427,Z 346.935,A -85,B 0,C 180,E1 -14469.865,E2 -14469.865} C_VEL
LIN {X 0,Y 337.691,Z 357.751,A -85,B 0,C 180,E1 -14471.495,E2 -14471.495} C_VEL
LIN {X 0,Y 336.154,Z 367.503,A -85,B 0,C 180,E1 -14473.293,E2 -14473.293} C_VEL
LIN {X 0,Y 335.069,Z 374.89,A -85,B 0,C 180,E1 -14474.933,E2 -14474.933} C_VEL
LIN {X 0,Y 333.969,Z 382.343,A -85,B 0,C 180,E1 -14476.925,E2 -14476.925} C_VEL
LIN {X 0,Y 332.969,Z 388.769,A -85,B 0,C 180,E1 -14479.049,E2 -14479.049} C_VEL
LIN {X 0,Y 332.357,Z 394.471,A -85,B 0,C 180,E1 -14481.488,E2 -14481.488} C_VEL
LIN {X 0,Y 332.043,Z 398.61,A -85,B 0,C 180,E1 -14483.925,E2 -14483.925} C_VEL
LIN {X 0,Y 331.945,Z 401.314,A -85,B 0,C 180,E1 -14486.358,E2 -14486.358} C_VEL
LIN {X 0,Y 331.868,Z 402.651,A -85,B 0,C 180,E1 -14488.786,E2 -14488.786} C_VEL
LIN {X 0,Y 331.868,Z 402.647,A -85,B 0,C 180,E1 -14491.213,E2 -14491.213} C_VEL
LIN {X 0,Y 331.944,Z 401.303,A -85,B 0,C 180,E1 -14493.642,E2 -14493.642} C_VEL
LIN {X 0,Y 332.043,Z 398.593,A -85,B 0,C 180,E1 -14496.075,E2 -14496.075} C_VEL
LIN {X 0,Y 332.356,Z 394.441,A -85,B 0,C 180,E1 -14498.512,E2 -14498.512} C_VEL
LIN {X 0,Y 332.968,Z 388.727,A -85,B 0,C 180,E1 -14500.951,E2 -14500.951} C_VEL
LIN {X 0,Y 333.953,Z 382.292,A -85,B 0,C 180,E1 -14503.075,E2 -14503.075} C_VEL
LIN {X 0,Y 335.08,Z 374.854,A -85,B 0,C 180,E1 -14505.059,E2 -14505.059} C_VEL
LIN {X 0,Y 336.369,Z 365.934,A -85,B 0,C 180,E1 -14507.008,E2 -14507.008} C_VEL
LIN {X 0,Y 337.977,Z 355.87,A -85,B 0,C 180,E1 -14508.803,E2 -14508.803} C_VEL
LIN {X 0,Y 339.741,Z 344.644,A -85,B 0,C 180,E1 -14510.431,E2 -14510.431} C_VEL
LIN {X 0,Y 341.423,Z 333.48,A -85,B 0,C 180,E1 -14511.748,E2 -14511.748} C_VEL
LIN {X 0,Y 343.02,Z 321.317,A -85,B 0,C 180,E1 -14512.91,E2 -14512.91} C_VEL
LIN {X 0,Y 343.146,Z 316.619,A -85,B 0,C 180,E1 -14513.324,E2 -14513.324} C_VEL
LIN {X 0,Y 341.241,Z 303.333,A -85,B 0,C 180,E1 -14514.477,E2 -14514.477} C_VEL
LIN {X 0,Y 338.382,Z 289.648,A -85,B 0,C 180,E1 -14515.486,E2 -14515.486} C_VEL
LIN {X 0,Y 334.245,Z 275.148,A -85,B 0,C 180,E1 -14516.394,E2 -14516.394} C_VEL
LIN {X 0,Y 333.293,Z 271.497,A -85,B 0,C 180,E1 -14516.597,E2 -14516.597} C_VEL
LIN {X 0,Y 333.817,Z 266.195,A -85,B 0,C 180,E1 -14520.35,E2 -14520.35} C_VEL
LIN {X 0,Y 334.174,Z 262.351,A -85,B 0,C 180,E1 -14523.148,E2 -14523.148} C_VEL
LIN {X 0,Y 334.772,Z 257.136,A -85,B 0,C 180,E1 -14527.084,E2 -14527.084} C_VEL
LIN {X 0,Y 334.934,Z 254.581,A -85,B 0,C 180,E1 -14529.07,E2 -14529.07} C_VEL
LIN {X 0,Y 334.793,Z 252.32,A -85,B 0,C 180,E1 -14530.912,E2 -14530.912} C_VEL
LIN {X 0,Y 334.261,Z 248.328,A -85,B 0,C 180,E1 -14534.368,E2 -14534.368} C_VEL
LIN {X 0,Y 333.698,Z 244.545,A -85,B 0,C 180,E1 -14538.034,E2 -14538.034} C_VEL
LIN {X 0,Y 333.652,Z 244.553,A -85,B 0,C 180,E1 -14542.349,E2 -14542.349} C_VEL
LIN {X 0,Y 333.675,Z 244.549,A -85,B 0,C 180,E1 -14545.341,E2 -14545.341} C_VEL
LIN {X 0,Y 333.63,Z 244.553,A -85,B 0,C 180,E1 -14548.222,E2 -14548.222} C_VEL
LIN {X 0,Y 333.655,Z 244.55,A -85,B 0,C 180,E1 -14551.023,E2 -14551.023} C_VEL
LIN {X 0,Y 333.697,Z 244.544,A -85,B 0,C 180,E1 -14555.088,E2 -14555.088} C_VEL
LIN {X 0,Y 333.674,Z 244.549,A -85,B 0,C 180,E1 -14559.019,E2 -14559.019} C_VEL
LIN {X 0,Y 333.742,Z 244.537,A -85,B 0,C 180,E1 -14561.587,E2 -14561.587} C_VEL
LIN {X 0,Y 333.809,Z 244.526,A -85,B 0,C 180,E1 -14565.577,E2 -14565.577} C_VEL
LIN {X 0,Y 333.819,Z 244.522,A -85,B 0,C 180,E1 -14569.078,E2 -14569.078} C_VEL
LIN {X 0,Y 333.959,Z 244.509,A -85,B 0,C 180,E1 -14572.746,E2 -14572.746} C_VEL
LIN {X 0,Y 333.8,Z 244.532,A -85,B 0,C 180,E1 -14575.169,E2 -14575.169} C_VEL
LIN {X 0,Y 334.106,Z 244.491,A -85,B 0,C 180,E1 -14577.589,E2 -14577.589} C_VEL
LIN {X 0,Y 334.189,Z 244.483,A -85,B 0,C 180,E1 -14580,E2 -14580} C_VEL
LIN {X 0,Y 334.102,Z 244.492,A -85,B 0,C 180,E1 -14582.411,E2 -14582.411} C_VEL
LIN {X 0,Y 333.992,Z 244.504,A -85,B 0,C 180,E1 -14586.683,E2 -14586.683} C_VEL
LIN {X 0,Y 333.853,Z 244.525,A -85,B 0,C 180,E1 -14589.695,E2 -14589.695} C_VEL
LIN {X 0,Y 333.798,Z 244.529,A -85,B 0,C 180,E1 -14593.391,E2 -14593.391} C_VEL
LIN {X 0,Y 333.748,Z 244.537,A -85,B 0,C 180,E1 -14597.146,E2 -14597.146} C_VEL
LIN {X 0,Y 333.736,Z 244.538,A -85,B 0,C 180,E1 -14599.69,E2 -14599.69} C_VEL
LIN {X 0,Y 333.671,Z 244.546,A -85,B 0,C 180,E1 -14603.59,E2 -14603.59} C_VEL
LIN {X 0,Y 333.736,Z 244.539,A -85,B 0,C 180,E1 -14606.246,E2 -14606.246} C_VEL
LIN {X 0,Y 333.691,Z 244.545,A -85,B 0,C 180,E1 -14608.974,E2 -14608.974} C_VEL
LIN {X 0,Y 333.645,Z 244.551,A -85,B 0,C 180,E1 -14612.587,E2 -14612.587} C_VEL
LIN {X 0,Y 333.676,Z 244.547,A -85,B 0,C 180,E1 -14616.139,E2 -14616.139} C_VEL
LIN {X 0,Y 333.621,Z 244.553,A -85,B 0,C 180,E1 -14619.196,E2 -14619.196} C_VEL
LIN {X 0,Y 333.63,Z 244.556,A -85,B 0,C 180,E1 -14622.499,E2 -14622.499} C_VEL
LIN {X 0,Y 333.597,Z 244.558,A -85,B 0,C 180,E1 -14625.955,E2 -14625.955} C_VEL
LIN {X 0,Y 333.658,Z 244.637,A -85,B 0,C 180,E1 -14627.621,E2 -14627.621} C_VEL
LIN {X 0,Y 333.928,Z 247.619,A -85,B 0,C 180,E1 -14630.847,E2 -14630.847} C_VEL
LIN {X 0,Y 333.831,Z 250.602,A -85,B 0,C 180,E1 -14633.88,E2 -14633.88} C_VEL
LIN {X 0,Y 333.52,Z 254.335,A -85,B 0,C 180,E1 -14637.447,E2 -14637.447} C_VEL
LIN {X 0,Y 333.177,Z 258.155,A -85,B 0,C 180,E1 -14640.977,E2 -14640.977} C_VEL
LIN {X 0,Y 333.023,Z 260.926,A -85,B 0,C 180,E1 -14643.464,E2 -14643.464} C_VEL
LIN {X 0,Y 334.889,Z 266.711,A -85,B 0,C 180,E1 -14643.8,E2 -14643.8} C_VEL
LIN {X 0,Y 339.156,Z 280.182,A -85,B 0,C 180,E1 -14644.732,E2 -14644.732} C_VEL
LIN {X 0,Y 342.277,Z 293.026,A -85,B 0,C 180,E1 -14645.754,E2 -14645.754} C_VEL
LIN {X 0,Y 344.029,Z 302.534,A -85,B 0,C 180,E1 -14646.609,E2 -14646.609} C_VEL
LIN {X 0,Y 343.048,Z 313.695,A -85,B 0,C 180,E1 -14647.57,E2 -14647.57} C_VEL
LIN {X 0,Y 341.387,Z 326.252,A -85,B 0,C 180,E1 -14648.884,E2 -14648.884} C_VEL
LIN {X 0,Y 339.666,Z 337.603,A -85,B 0,C 180,E1 -14650.353,E2 -14650.353} C_VEL
LIN {X 0,Y 338.14,Z 347.009,A -85,B 0,C 180,E1 -14651.834,E2 -14651.834} C_VEL
LIN {X 0,Y 336.558,Z 356.461,A -85,B 0,C 180,E1 -14653.627,E2 -14653.627} C_VEL
LIN {X 0,Y 335.413,Z 364.282,A -85,B 0,C 180,E1 -14655.437,E2 -14655.437} C_VEL
LIN {X 0,Y 334.247,Z 370.793,A -85,B 0,C 180,E1 -14657.245,E2 -14657.245} C_VEL
LIN {X 0,Y 333.458,Z 376.193,A -85,B 0,C 180,E1 -14659.066,E2 -14659.066} C_VEL
LIN {X 0,Y 332.709,Z 381.868,A -85,B 0,C 180,E1 -14661.497,E2 -14661.497} C_VEL
LIN {X 0,Y 332.289,Z 385.991,A -85,B 0,C 180,E1 -14663.93,E2 -14663.93} C_VEL
LIN {X 0,Y 332.049,Z 388.687,A -85,B 0,C 180,E1 -14666.36,E2 -14666.36} C_VEL
LIN {X 0,Y 331.895,Z 390.038,A -85,B 0,C 180,E1 -14668.787,E2 -14668.787} C_VEL
LIN {X 0,Y 331.895,Z 390.07,A -85,B 0,C 180,E1 -14671.213,E2 -14671.213} C_VEL
LIN {X 0,Y 332.047,Z 388.78,A -85,B 0,C 180,E1 -14673.641,E2 -14673.641} C_VEL
LIN {X 0,Y 332.289,Z 386.14,A -85,B 0,C 180,E1 -14676.071,E2 -14676.071} C_VEL
LIN {X 0,Y 332.703,Z 382.081,A -85,B 0,C 180,E1 -14678.504,E2 -14678.504} C_VEL
LIN {X 0,Y 333.42,Z 376.471,A -85,B 0,C 180,E1 -14680.936,E2 -14680.936} C_VEL
LIN {X 0,Y 334.399,Z 370.134,A -85,B 0,C 180,E1 -14683.058,E2 -14683.058} C_VEL
LIN {X 0,Y 335.628,Z 362.592,A -85,B 0,C 180,E1 -14685.088,E2 -14685.088} C_VEL
LIN {X 0,Y 336.711,Z 355.485,A -85,B 0,C 180,E1 -14686.678,E2 -14686.678} C_VEL
LIN {X 0,Y 338.392,Z 345.838,A -85,B 0,C 180,E1 -14688.465,E2 -14688.465} C_VEL
LIN {X 0,Y 340.056,Z 335.132,A -85,B 0,C 180,E1 -14690.096,E2 -14690.096} C_VEL
LIN {X 0,Y 341.81,Z 323.262,A -85,B 0,C 180,E1 -14691.564,E2 -14691.564} C_VEL
LIN {X 0,Y 343.305,Z 311.514,A -85,B 0,C 180,E1 -14692.739,E2 -14692.739} C_VEL
LIN {X 0,Y 344.17,Z 303.103,A -85,B 0,C 180,E1 -14693.443,E2 -14693.443} C_VEL
LIN {X 0,Y 341.585,Z 289.723,A -85,B 0,C 180,E1 -14694.63,E2 -14694.63} C_VEL
LIN {X 0,Y 338.122,Z 276.655,A -85,B 0,C 180,E1 -14695.636,E2 -14695.636} C_VEL
LIN {X 0,Y 333.69,Z 263.423,A -85,B 0,C 180,E1 -14696.518,E2 -14696.518} C_VEL
LIN {X 0,Y 333.023,Z 260.896,A -85,B 0,C 180,E1 -14696.677,E2 -14696.677} C_VEL
LIN {X 0,Y 333.299,Z 256.777,A -85,B 0,C 180,E1 -14700.402,E2 -14700.402} C_VEL
LIN {X 0,Y 333.575,Z 253.752,A -85,B 0,C 180,E1 -14703.216,E2 -14703.216} C_VEL
LIN {X 0,Y 333.832,Z 250.722,A -85,B 0,C 180,E1 -14706.12,E2 -14706.12} C_VEL
LIN {X 0,Y 333.915,Z 247.728,A -85,B 0,C 180,E1 -14709.155,E2 -14709.155} C_VEL
LIN {X 0,Y 333.635,Z 244.649,A -85,B 0,C 180,E1 -14712.5,E2 -14712.5} C_VEL
LIN {X 0,Y 333.591,Z 244.56,A -85,B 0,C 180,E1 -14716.087,E2 -14716.087} C_VEL
LIN {X 0,Y 332.91,Z 244.645,A -85,B 0,C 180,E1 -14717.095,E2 -14717.095} C_VEL
LIN {X 0,Y 330.089,Z 244.996,A -85,B 0,C 180,E1 -14718.736,E2 -14718.736} C_VEL
LIN {X 0,Y 327.705,Z 245.296,A -85,B 0,C 180,E1 -14720.064,E2 -14720.064} C_VEL
LIN {X 0,Y 326.672,Z 245.422,A -85,B 0,C 180,E1 -14721.092,E2 -14721.092} C_VEL
LIN {X 0,Y 326.582,Z 245.431,A -85,B 0,C 180,E1 -14721.44,E2 -14721.44} C_VEL
LIN {X 0,Y 326.621,Z 245.425,A -85,B 0,C 180,E1 -14724.851,E2 -14724.851} C_VEL
LIN {X 0,Y 326.61,Z 245.428,A -85,B 0,C 180,E1 -14727.456,E2 -14727.456} C_VEL
LIN {X 0,Y 326.65,Z 245.422,A -85,B 0,C 180,E1 -14730.34,E2 -14730.34} C_VEL
LIN {X 0,Y 326.692,Z 245.411,A -85,B 0,C 180,E1 -14734.516,E2 -14734.516} C_VEL
LIN {X 0,Y 326.622,Z 245.425,A -85,B 0,C 180,E1 -14738.543,E2 -14738.543} C_VEL
LIN {X 0,Y 326.747,Z 245.409,A -85,B 0,C 180,E1 -14741.178,E2 -14741.178} C_VEL
LIN {X 0,Y 326.766,Z 245.409,A -85,B 0,C 180,E1 -14745.433,E2 -14745.433} C_VEL
LIN {X 0,Y 326.761,Z 245.407,A -85,B 0,C 180,E1 -14748.839,E2 -14748.839} C_VEL
LIN {X 0,Y 326.945,Z 245.384,A -85,B 0,C 180,E1 -14752.589,E2 -14752.589} C_VEL
LIN {X 0,Y 326.985,Z 245.379,A -85,B 0,C 180,E1 -14753.831,E2 -14753.831} C_VEL
LIN {X 0,Y 327.044,Z 245.37,A -85,B 0,C 180,E1 -14757.537,E2 -14757.537} C_VEL
LIN {X 0,Y 327.056,Z 245.371,A -85,B 0,C 180,E1 -14761.231,E2 -14761.231} C_VEL
LIN {X 0,Y 327.047,Z 245.369,A -85,B 0,C 180,E1 -14762.463,E2 -14762.463} C_VEL
LIN {X 0,Y 326.948,Z 245.385,A -85,B 0,C 180,E1 -14766.17,E2 -14766.17} C_VEL
LIN {X 0,Y 326.786,Z 245.405,A -85,B 0,C 180,E1 -14769.907,E2 -14769.907} C_VEL
LIN {X 0,Y 326.762,Z 245.408,A -85,B 0,C 180,E1 -14773.685,E2 -14773.685} C_VEL
LIN {X 0,Y 326.667,Z 245.42,A -85,B 0,C 180,E1 -14777.53,E2 -14777.53} C_VEL
LIN {X 0,Y 326.652,Z 245.421,A -85,B 0,C 180,E1 -14780.136,E2 -14780.136} C_VEL
LIN {X 0,Y 326.634,Z 245.425,A -85,B 0,C 180,E1 -14784.13,E2 -14784.13} C_VEL
LIN {X 0,Y 326.603,Z 245.427,A -85,B 0,C 180,E1 -14788.084,E2 -14788.084} C_VEL
LIN {X 0,Y 326.575,Z 245.429,A -85,B 0,C 180,E1 -14791.097,E2 -14791.097} C_VEL
LIN {X 0,Y 326.609,Z 245.428,A -85,B 0,C 180,E1 -14794.019,E2 -14794.019} C_VEL
LIN {X 0,Y 326.629,Z 245.429,A -85,B 0,C 180,E1 -14797.238,E2 -14797.238} C_VEL
LIN {X 0,Y 326.601,Z 245.431,A -85,B 0,C 180,E1 -14801.136,E2 -14801.136} C_VEL
LIN {X 0,Y 326.663,Z 245.602,A -85,B 0,C 180,E1 -14801.832,E2 -14801.832} C_VEL
LIN {X 0,Y 327.208,Z 249.072,A -85,B 0,C 180,E1 -14805.137,E2 -14805.137} C_VEL
LIN {X 0,Y 327.735,Z 252.999,A -85,B 0,C 180,E1 -14808.638,E2 -14808.638} C_VEL
LIN {X 0,Y 327.851,Z 256.51,A -85,B 0,C 180,E1 -14811.562,E2 -14811.562} C_VEL
LIN {X 0,Y 327.475,Z 260.421,A -85,B 0,C 180,E1 -14814.639,E2 -14814.639} C_VEL
LIN {X 0,Y 327.046,Z 264.174,A -85,B 0,C 180,E1 -14817.504,E2 -14817.504} C_VEL
LIN {X 0,Y 326.632,Z 267.997,A -85,B 0,C 180,E1 -14820.338,E2 -14820.338} C_VEL
LIN {X 0,Y 326.337,Z 271.357,A -85,B 0,C 180,E1 -14822.764,E2 -14822.764} C_VEL
LIN {X 0,Y 331.179,Z 288.44,A -85,B 0,C 180,E1 -14823.848,E2 -14823.848} C_VEL
LIN {X 0,Y 334.264,Z 302.236,A -85,B 0,C 180,E1 -14824.895,E2 -14824.895} C_VEL
LIN {X 0,Y 336.289,Z 315.381,A -85,B 0,C 180,E1 -14826.056,E2 -14826.056} C_VEL
LIN {X 0,Y 336.6,Z 319.895,A -85,B 0,C 180,E1 -14826.491,E2 -14826.491} C_VEL
LIN {X 0,Y 334.997,Z 332.471,A -85,B 0,C 180,E1 -14827.696,E2 -14827.696} C_VEL
LIN {X 0,Y 333.088,Z 344.638,A -85,B 0,C 180,E1 -14829.142,E2 -14829.142} C_VEL
LIN {X 0,Y 331.252,Z 355.832,A -85,B 0,C 180,E1 -14830.8,E2 -14830.8} C_VEL
LIN {X 0,Y 329.559,Z 365.878,A -85,B 0,C 180,E1 -14832.629,E2 -14832.629} C_VEL
LIN {X 0,Y 328.084,Z 375.354,A -85,B 0,C 180,E1 -14834.759,E2 -14834.759} C_VEL
LIN {X 0,Y 326.838,Z 383.22,A -85,B 0,C 180,E1 -14836.951,E2 -14836.951} C_VEL
LIN {X 0,Y 325.949,Z 388.635,A -85,B 0,C 180,E1 -14838.81,E2 -14838.81} C_VEL
LIN {X 0,Y 325.311,Z 394.337,A -85,B 0,C 180,E1 -14841.302,E2 -14841.302} C_VEL
LIN {X 0,Y 324.959,Z 398.475,A -85,B 0,C 180,E1 -14843.792,E2 -14843.792} C_VEL
LIN {X 0,Y 324.853,Z 401.179,A -85,B 0,C 180,E1 -14846.279,E2 -14846.279} C_VEL
LIN {X 0,Y 324.779,Z 402.516,A -85,B 0,C 180,E1 -14848.76,E2 -14848.76} C_VEL
LIN {X 0,Y 324.779,Z 402.512,A -85,B 0,C 180,E1 -14851.24,E2 -14851.24} C_VEL
LIN {X 0,Y 324.852,Z 401.168,A -85,B 0,C 180,E1 -14853.721,E2 -14853.721} C_VEL
LIN {X 0,Y 324.959,Z 398.457,A -85,B 0,C 180,E1 -14856.208,E2 -14856.208} C_VEL
LIN {X 0,Y 325.309,Z 394.305,A -85,B 0,C 180,E1 -14858.698,E2 -14858.698} C_VEL
LIN {X 0,Y 325.948,Z 388.59,A -85,B 0,C 180,E1 -14861.189,E2 -14861.189} C_VEL
LIN {X 0,Y 327.005,Z 382.155,A -85,B 0,C 180,E1 -14863.358,E2 -14863.358} C_VEL
LIN {X 0,Y 328.186,Z 374.285,A -85,B 0,C 180,E1 -14865.494,E2 -14865.494} C_VEL
LIN {X 0,Y 329.546,Z 365.796,A -85,B 0,C 180,E1 -14867.372,E2 -14867.372} C_VEL
LIN {X 0,Y 331.243,Z 355.733,A -85,B 0,C 180,E1 -14869.2,E2 -14869.2} C_VEL
LIN {X 0,Y 333.084,Z 344.506,A -85,B 0,C 180,E1 -14870.858,E2 -14870.858} C_VEL
LIN {X 0,Y 335.046,Z 331.959,A -85,B 0,C 180,E1 -14872.34,E2 -14872.34} C_VEL
LIN {X 0,Y 336.578,Z 319.709,A -85,B 0,C 180,E1 -14873.509,E2 -14873.509} C_VEL
LIN {X 0,Y 335.44,Z 309.589,A -85,B 0,C 180,E1 -14874.463,E2 -14874.463} C_VEL
LIN {X 0,Y 333.245,Z 297.161,A -85,B 0,C 180,E1 -14875.49,E2 -14875.49} C_VEL
LIN {X 0,Y 329.689,Z 282.965,A -85,B 0,C 180,E1 -14876.506,E2 -14876.506} C_VEL
LIN {X 0,Y 326.327,Z 271.5,A -85,B 0,C 180,E1 -14877.185,E2 -14877.185} C_VEL
LIN {X 0,Y 326.835,Z 266.046,A -85,B 0,C 180,E1 -14881.069,E2 -14881.069} C_VEL
LIN {X 0,Y 327.216,Z 262.232,A -85,B 0,C 180,E1 -14883.947,E2 -14883.947} C_VEL
LIN {X 0,Y 327.808,Z 257.636,A -85,B 0,C 180,E1 -14887.509,E2 -14887.509} C_VEL
LIN {X 0,Y 327.86,Z 254.534,A -85,B 0,C 180,E1 -14890.022,E2 -14890.022} C_VEL
LIN {X 0,Y 327.432,Z 250.652,A -85,B 0,C 180,E1 -14893.381,E2 -14893.381} C_VEL
LIN {X 0,Y 326.828,Z 246.768,A -85,B 0,C 180,E1 -14896.981,E2 -14896.981} C_VEL
LIN {X 0,Y 326.633,Z 245.426,A -85,B 0,C 180,E1 -14898.366,E2 -14898.366} C_VEL
LIN {X 0,Y 326.624,Z 245.428,A -85,B 0,C 180,E1 -14901.391,E2 -14901.391} C_VEL
LIN {X 0,Y 326.62,Z 245.428,A -85,B 0,C 180,E1 -14904.851,E2 -14904.851} C_VEL
LIN {X 0,Y 326.608,Z 245.43,A -85,B 0,C 180,E1 -14907.456,E2 -14907.456} C_VEL
LIN {X 0,Y 326.617,Z 245.426,A -85,B 0,C 180,E1 -14910.337,E2 -14910.337} C_VEL
LIN {X 0,Y 326.642,Z 245.423,A -85,B 0,C 180,E1 -14914.645,E2 -14914.645} C_VEL
LIN {X 0,Y 326.62,Z 245.426,A -85,B 0,C 180,E1 -14918.544,E2 -14918.544} C_VEL
LIN {X 0,Y 326.708,Z 245.413,A -85,B 0,C 180,E1 -14921.175,E2 -14921.175} C_VEL
LIN {X 0,Y 326.764,Z 245.404,A -85,B 0,C 180,E1 -14925.433,E2 -14925.433} C_VEL
LIN {X 0,Y 326.759,Z 245.403,A -85,B 0,C 180,E1 -14928.839,E2 -14928.839} C_VEL
LIN {X 0,Y 326.915,Z 245.386,A -85,B 0,C 180,E1 -14932.589,E2 -14932.589} C_VEL
LIN {X 0,Y 326.767,Z 245.407,A -85,B 0,C 180,E1 -14935.065,E2 -14935.065} C_VEL
LIN {X 0,Y 327.046,Z 245.371,A -85,B 0,C 180,E1 -14937.537,E2 -14937.537} C_VEL
LIN {X 0,Y 327.142,Z 245.361,A -85,B 0,C 180,E1 -14940,E2 -14940} C_VEL
LIN {X 0,Y 327.043,Z 245.371,A -85,B 0,C 180,E1 -14942.463,E2 -14942.463} C_VEL
LIN {X 0,Y 326.959,Z 245.381,A -85,B 0,C 180,E1 -14946.676,E2 -14946.676} C_VEL
LIN {X 0,Y 326.808,Z 245.403,A -85,B 0,C 180,E1 -14949.907,E2 -14949.907} C_VEL
LIN {X 0,Y 326.761,Z 245.405,A -85,B 0,C 180,E1 -14953.685,E2 -14953.685} C_VEL
LIN {X 0,Y 326.701,Z 245.416,A -85,B 0,C 180,E1 -14957.528,E2 -14957.528} C_VEL
LIN {X 0,Y 326.662,Z 245.418,A -85,B 0,C 180,E1 -14960.135,E2 -14960.135} C_VEL
LIN {X 0,Y 326.65,Z 245.421,A -85,B 0,C 180,E1 -14964.129,E2 -14964.129} C_VEL
LIN {X 0,Y 326.684,Z 245.416,A -85,B 0,C 180,E1 -14966.858,E2 -14966.858} C_VEL
LIN {X 0,Y 326.635,Z 245.424,A -85,B 0,C 180,E1 -14970.61,E2 -14970.61} C_VEL
LIN {X 0,Y 326.608,Z 245.428,A -85,B 0,C 180,E1 -14974.019,E2 -14974.019} C_VEL
LIN {X 0,Y 326.624,Z 245.426,A -85,B 0,C 180,E1 -14977.238,E2 -14977.238} C_VEL
LIN {X 0,Y 326.545,Z 245.436,A -85,B 0,C 180,E1 -14981.125,E2 -14981.125} C_VEL
LIN {X 0,Y 326.562,Z 245.434,A -85,B 0,C 180,E1 -14983.526,E2 -14983.526} C_VEL
LIN {X 0,Y 326.581,Z 245.433,A -85,B 0,C 180,E1 -14987.027,E2 -14987.027} C_VEL
LIN {X 0,Y 326.821,Z 247.736,A -85,B 0,C 180,E1 -14989.825,E2 -14989.825} C_VEL
LIN {X 0,Y 326.832,Z 250.731,A -85,B 0,C 180,E1 -14992.98,E2 -14992.98} C_VEL
LIN {X 0,Y 326.607,Z 253.749,A -85,B 0,C 180,E1 -14995.981,E2 -14995.981} C_VEL
LIN {X 0,Y 326.263,Z 257.457,A -85,B 0,C 180,E1 -14999.501,E2 -14999.501} C_VEL
LIN {X 0,Y 326.016,Z 261.046,A -85,B 0,C 180,E1 -15002.831,E2 -15002.831} C_VEL
LIN {X 0,Y 327.978,Z 267.032,A -85,B 0,C 180,E1 -15003.21,E2 -15003.21} C_VEL
LIN {X 0,Y 332.271,Z 280.446,A -85,B 0,C 180,E1 -15004.176,E2 -15004.176} C_VEL
LIN {X 0,Y 335.421,Z 293.177,A -85,B 0,C 180,E1 -15005.225,E2 -15005.225} C_VEL
LIN {X 0,Y 337.287,Z 303.079,A -85,B 0,C 180,E1 -15006.145,E2 -15006.145} C_VEL
LIN {X 0,Y 337.289,Z 306.652,A -85,B 0,C 180,E1 -15006.466,E2 -15006.466} C_VEL
LIN {X 0,Y 335.712,Z 319.834,A -85,B 0,C 180,E1 -15007.711,E2 -15007.711} C_VEL
LIN {X 0,Y 333.976,Z 331.182,A -85,B 0,C 180,E1 -15009.039,E2 -15009.039} C_VEL
LIN {X 0,Y 332.342,Z 341.677,A -85,B 0,C 180,E1 -15010.545,E2 -15010.545} C_VEL
LIN {X 0,Y 330.527,Z 352.099,A -85,B 0,C 180,E1 -15012.362,E2 -15012.362} C_VEL
LIN {X 0,Y 328.943,Z 360.809,A -85,B 0,C 180,E1 -15014.22,E2 -15014.22} C_VEL
LIN {X 0,Y 327.935,Z 367.824,A -85,B 0,C 180,E1 -15016.049,E2 -15016.049} C_VEL
LIN {X 0,Y 326.719,Z 374.657,A -85,B 0,C 180,E1 -15018.208,E2 -15018.208} C_VEL
LIN {X 0,Y 326.028,Z 379.37,A -85,B 0,C 180,E1 -15020.07,E2 -15020.07} C_VEL
LIN {X 0,Y 325.403,Z 384.251,A -85,B 0,C 180,E1 -15022.554,E2 -15022.554} C_VEL
LIN {X 0,Y 325.064,Z 387.647,A -85,B 0,C 180,E1 -15025.039,E2 -15025.039} C_VEL
LIN {X 0,Y 324.862,Z 389.663,A -85,B 0,C 180,E1 -15027.52,E2 -15027.52} C_VEL
LIN {X 0,Y 324.811,Z 390.353,A -85,B 0,C 180,E1 -15030,E2 -15030} C_VEL
LIN {X 0,Y 324.861,Z 389.726,A -85,B 0,C 180,E1 -15032.48,E2 -15032.48} C_VEL
LIN {X 0,Y 325.062,Z 387.766,A -85,B 0,C 180,E1 -15034.961,E2 -15034.961} C_VEL
LIN {X 0,Y 325.402,Z 384.429,A -85,B 0,C 180,E1 -15037.446,E2 -15037.446} C_VEL
LIN {X 0,Y 326.011,Z 379.614,A -85,B 0,C 180,E1 -15039.931,E2 -15039.931} C_VEL
LIN {X 0,Y 326.67,Z 374.966,A -85,B 0,C 180,E1 -15041.794,E2 -15041.794} C_VEL
LIN {X 0,Y 327.88,Z 368.201,A -85,B 0,C 180,E1 -15043.954,E2 -15043.954} C_VEL
LIN {X 0,Y 328.827,Z 361.567,A -85,B 0,C 180,E1 -15045.708,E2 -15045.708} C_VEL
LIN {X 0,Y 330.424,Z 352.644,A -85,B 0,C 180,E1 -15047.644,E2 -15047.644} C_VEL
LIN {X 0,Y 332.212,Z 342.335,A -85,B 0,C 180,E1 -15049.463,E2 -15049.463} C_VEL
LIN {X 0,Y 334.15,Z 330.798,A -85,B 0,C 180,E1 -15051.112,E2 -15051.112} C_VEL
LIN {X 0,Y 335.778,Z 319.611,A -85,B 0,C 180,E1 -15052.418,E2 -15052.418} C_VEL
LIN {X 0,Y 337.304,Z 307.027,A -85,B 0,C 180,E1 -15053.608,E2 -15053.608} C_VEL
LIN {X 0,Y 337.405,Z 303.887,A -85,B 0,C 180,E1 -15053.888,E2 -15053.888} C_VEL
LIN {X 0,Y 335.048,Z 291.253,A -85,B 0,C 180,E1 -15055.054,E2 -15055.054} C_VEL
LIN {X 0,Y 331.413,Z 277.398,A -85,B 0,C 180,E1 -15056.165,E2 -15056.165} C_VEL
LIN {X 0,Y 326.76,Z 263.711,A -85,B 0,C 180,E1 -15057.121,E2 -15057.121} C_VEL
LIN {X 0,Y 326.039,Z 261.065,A -85,B 0,C 180,E1 -15057.263,E2 -15057.263} C_VEL
LIN {X 0,Y 326.293,Z 256.911,A -85,B 0,C 180,E1 -15061.127,E2 -15061.127} C_VEL
LIN {X 0,Y 326.612,Z 253.87,A -85,B 0,C 180,E1 -15064.019,E2 -15064.019} C_VEL
LIN {X 0,Y 326.833,Z 250.59,A -85,B 0,C 180,E1 -15067.286,E2 -15067.286} C_VEL
LIN {X 0,Y 326.817,Z 247.849,A -85,B 0,C 180,E1 -15070.176,E2 -15070.176} C_VEL
LIN {X 0,Y 326.555,Z 245.435,A -85,B 0,C 180,E1 -15072.968,E2 -15072.968} C_VEL
LIN {X 0,Y 326.576,Z 245.434,A -85,B 0,C 180,E1 -15077.029,E2 -15077.029} C_VEL
LIN {X 0,Y 326.584,Z 245.431,A -85,B 0,C 180,E1 -15081.386,E2 -15081.386} C_VEL
LIN {X 0,Y 326.582,Z 245.431,A -85,B 0,C 180,E1 -15081.44,E2 -15081.44} C_VEL
LIN {X 0,Y 325.914,Z 245.514,A -85,B 0,C 180,E1 -15082.47,E2 -15082.47} C_VEL
LIN {X 0,Y 323.114,Z 245.863,A -85,B 0,C 180,E1 -15084.147,E2 -15084.147} C_VEL
LIN {X 0,Y 320.724,Z 246.162,A -85,B 0,C 180,E1 -15085.506,E2 -15085.506} C_VEL
LIN {X 0,Y 319.664,Z 246.292,A -85,B 0,C 180,E1 -15086.556,E2 -15086.556} C_VEL
LIN {X 0,Y 319.559,Z 246.303,A -85,B 0,C 180,E1 -15086.912,E2 -15086.912} C_VEL
LIN {X 0,Y 319.587,Z 246.302,A -85,B 0,C 180,E1 -15089.616,E2 -15089.616} C_VEL
LIN {X 0,Y 319.608,Z 246.3,A -85,B 0,C 180,E1 -15092.498,E2 -15092.498} C_VEL
LIN {X 0,Y 319.605,Z 246.294,A -85,B 0,C 180,E1 -15095.304,E2 -15095.304} C_VEL
LIN {X 0,Y 319.605,Z 246.298,A -85,B 0,C 180,E1 -15099.4,E2 -15099.4} C_VEL
LIN {X 0,Y 319.661,Z 246.292,A -85,B 0,C 180,E1 -15102.073,E2 -15102.073} C_VEL
LIN {X 0,Y 319.735,Z 246.282,A -85,B 0,C 180,E1 -15106.008,E2 -15106.008} C_VEL
LIN {X 0,Y 319.738,Z 246.281,A -85,B 0,C 180,E1 -15109.872,E2 -15109.872} C_VEL
LIN {X 0,Y 319.938,Z 246.258,A -85,B 0,C 180,E1 -15113.694,E2 -15113.694} C_VEL
LIN {X 0,Y 319.988,Z 246.249,A -85,B 0,C 180,E1 -15117.482,E2 -15117.482} C_VEL
LIN {X 0,Y 320.024,Z 246.247,A -85,B 0,C 180,E1 -15121.258,E2 -15121.258} C_VEL
LIN {X 0,Y 319.739,Z 246.282,A -85,B 0,C 180,E1 -15123.781,E2 -15123.781} C_VEL
LIN {X 0,Y 319.904,Z 246.263,A -85,B 0,C 180,E1 -15126.306,E2 -15126.306} C_VEL
LIN {X 0,Y 319.738,Z 246.283,A -85,B 0,C 180,E1 -15130.128,E2 -15130.128} C_VEL
LIN {X 0,Y 319.735,Z 246.283,A -85,B 0,C 180,E1 -15133.992,E2 -15133.992} C_VEL
LIN {X 0,Y 319.627,Z 246.299,A -85,B 0,C 180,E1 -15137.929,E2 -15137.929} C_VEL
LIN {X 0,Y 319.599,Z 246.3,A -85,B 0,C 180,E1 -15140.6,E2 -15140.6} C_VEL
LIN {X 0,Y 319.554,Z 246.305,A -85,B 0,C 180,E1 -15143.321,E2 -15143.321} C_VEL
LIN {X 0,Y 319.571,Z 246.299,A -85,B 0,C 180,E1 -15146.094,E2 -15146.094} C_VEL
LIN {X 0,Y 319.545,Z 246.307,A -85,B 0,C 180,E1 -15148.938,E2 -15148.938} C_VEL
LIN {X 0,Y 319.526,Z 246.308,A -85,B 0,C 180,E1 -15151.862,E2 -15151.862} C_VEL
LIN {X 0,Y 319.582,Z 246.307,A -85,B 0,C 180,E1 -15155.543,E2 -15155.543} C_VEL
LIN {X 0,Y 319.559,Z 246.308,A -85,B 0,C 180,E1 -15158.01,E2 -15158.01} C_VEL
LIN {X 0,Y 319.569,Z 246.378,A -85,B 0,C 180,E1 -15161.282,E2 -15161.282} C_VEL
LIN {X 0,Y 320.146,Z 249.771,A -85,B 0,C 180,E1 -15164.626,E2 -15164.626} C_VEL
LIN {X 0,Y 320.672,Z 253.617,A -85,B 0,C 180,E1 -15168.173,E2 -15168.173} C_VEL
LIN {X 0,Y 320.886,Z 256.389,A -85,B 0,C 180,E1 -15170.568,E2 -15170.568} C_VEL
LIN {X 0,Y 320.8,Z 258.313,A -85,B 0,C 180,E1 -15172.163,E2 -15172.163} C_VEL
LIN {X 0,Y 320.315,Z 262.132,A -85,B 0,C 180,E1 -15175.217,E2 -15175.217} C_VEL
LIN {X 0,Y 319.791,Z 267.028,A -85,B 0,C 180,E1 -15178.992,E2 -15178.992} C_VEL
LIN {X 0,Y 319.348,Z 271.208,A -85,B 0,C 180,E1 -15182.117,E2 -15182.117} C_VEL
LIN {X 0,Y 324.205,Z 288.067,A -85,B 0,C 180,E1 -15183.23,E2 -15183.23} C_VEL
LIN {X 0,Y 327.205,Z 301.084,A -85,B 0,C 180,E1 -15184.248,E2 -15184.248} C_VEL
LIN {X 0,Y 329.319,Z 314.19,A -85,B 0,C 180,E1 -15185.428,E2 -15185.428} C_VEL
LIN {X 0,Y 329.935,Z 321.248,A -85,B 0,C 180,E1 -15186.126,E2 -15186.126} C_VEL
LIN {X 0,Y 328.244,Z 333.367,A -85,B 0,C 180,E1 -15187.331,E2 -15187.331} C_VEL
LIN {X 0,Y 326.25,Z 345.598,A -85,B 0,C 180,E1 -15188.849,E2 -15188.849} C_VEL
LIN {X 0,Y 324.532,Z 355.7,A -85,B 0,C 180,E1 -15190.387,E2 -15190.387} C_VEL
LIN {X 0,Y 322.744,Z 365.745,A -85,B 0,C 180,E1 -15192.25,E2 -15192.25} C_VEL
LIN {X 0,Y 321.212,Z 374.757,A -85,B 0,C 180,E1 -15194.303,E2 -15194.303} C_VEL
LIN {X 0,Y 320.06,Z 382.074,A -85,B 0,C 180,E1 -15196.346,E2 -15196.346} C_VEL
LIN {X 0,Y 318.936,Z 388.5,A -85,B 0,C 180,E1 -15198.561,E2 -15198.561} C_VEL
LIN {X 0,Y 318.277,Z 394.203,A -85,B 0,C 180,E1 -15201.108,E2 -15201.108} C_VEL
LIN {X 0,Y 317.886,Z 398.341,A -85,B 0,C 180,E1 -15203.653,E2 -15203.653} C_VEL
LIN {X 0,Y 317.764,Z 401.045,A -85,B 0,C 180,E1 -15206.195,E2 -15206.195} C_VEL
LIN {X 0,Y 317.693,Z 402.382,A -85,B 0,C 180,E1 -15208.732,E2 -15208.732} C_VEL
LIN {X 0,Y 317.693,Z 402.377,A -85,B 0,C 180,E1 -15211.267,E2 -15211.267} C_VEL
LIN {X 0,Y 317.763,Z 401.033,A -85,B 0,C 180,E1 -15213.804,E2 -15213.804} C_VEL
LIN {X 0,Y 317.886,Z 398.321,A -85,B 0,C 180,E1 -15216.347,E2 -15216.347} C_VEL
LIN {X 0,Y 318.247,Z 394.169,A -85,B 0,C 180,E1 -15218.893,E2 -15218.893} C_VEL
LIN {X 0,Y 318.934,Z 388.453,A -85,B 0,C 180,E1 -15221.439,E2 -15221.439} C_VEL
LIN {X 0,Y 320.05,Z 382.017,A -85,B 0,C 180,E1 -15223.654,E2 -15223.654} C_VEL
LIN {X 0,Y 321.182,Z 374.763,A -85,B 0,C 180,E1 -15225.678,E2 -15225.678} C_VEL
LIN {X 0,Y 322.733,Z 365.658,A -85,B 0,C 180,E1 -15227.75,E2 -15227.75} C_VEL
LIN {X 0,Y 324.521,Z 355.595,A -85,B 0,C 180,E1 -15229.614,E2 -15229.614} C_VEL
LIN {X 0,Y 326.432,Z 344.367,A -85,B 0,C 180,E1 -15231.304,E2 -15231.304} C_VEL
LIN {X 0,Y 328.247,Z 333.201,A -85,B 0,C 180,E1 -15232.668,E2 -15232.668} C_VEL
LIN {X 0,Y 329.919,Z 321.036,A -85,B 0,C 180,E1 -15233.875,E2 -15233.875} C_VEL
LIN {X 0,Y 328.797,Z 310.502,A -85,B 0,C 180,E1 -15234.903,E2 -15234.903} C_VEL
LIN {X 0,Y 326.543,Z 297.793,A -85,B 0,C 180,E1 -15236,E2 -15236} C_VEL
LIN {X 0,Y 322.915,Z 283.189,A -85,B 0,C 180,E1 -15237.091,E2 -15237.091} C_VEL
LIN {X 0,Y 319.442,Z 271.917,A -85,B 0,C 180,E1 -15237.804,E2 -15237.804} C_VEL
LIN {X 0,Y 319.347,Z 271.177,A -85,B 0,C 180,E1 -15237.883,E2 -15237.883} C_VEL
LIN {X 0,Y 319.869,Z 265.929,A -85,B 0,C 180,E1 -15241.824,E2 -15241.824} C_VEL
LIN {X 0,Y 320.44,Z 260.864,A -85,B 0,C 180,E1 -15245.758,E2 -15245.758} C_VEL
LIN {X 0,Y 320.793,Z 258.158,A -85,B 0,C 180,E1 -15247.936,E2 -15247.936} C_VEL
LIN {X 0,Y 320.869,Z 255.734,A -85,B 0,C 180,E1 -15249.95,E2 -15249.95} C_VEL
LIN {X 0,Y 320.507,Z 252.478,A -85,B 0,C 180,E1 -15252.825,E2 -15252.825} C_VEL
LIN {X 0,Y 319.955,Z 248.582,A -85,B 0,C 180,E1 -15256.458,E2 -15256.458} C_VEL
LIN {X 0,Y 319.556,Z 246.307,A -85,B 0,C 180,E1 -15258.926,E2 -15258.926} C_VEL
LIN {X 0,Y 319.562,Z 246.308,A -85,B 0,C 180,E1 -15262.348,E2 -15262.348} C_VEL
LIN {X 0,Y 319.561,Z 246.307,A -85,B 0,C 180,E1 -15265.123,E2 -15265.123} C_VEL
LIN {X 0,Y 319.525,Z 246.311,A -85,B 0,C 180,E1 -15268.137,E2 -15268.137} C_VEL
LIN {X 0,Y 319.572,Z 246.303,A -85,B 0,C 180,E1 -15271.603,E2 -15271.603} C_VEL
LIN {X 0,Y 319.574,Z 246.304,A -85,B 0,C 180,E1 -15275.302,E2 -15275.302} C_VEL
LIN {X 0,Y 319.568,Z 246.304,A -85,B 0,C 180,E1 -15278.046,E2 -15278.046} C_VEL
LIN {X 0,Y 319.658,Z 246.292,A -85,B 0,C 180,E1 -15280.979,E2 -15280.979} C_VEL
LIN {X 0,Y 319.714,Z 246.283,A -85,B 0,C 180,E1 -15285.288,E2 -15285.288} C_VEL
LIN {X 0,Y 319.716,Z 246.282,A -85,B 0,C 180,E1 -15288.59,E2 -15288.59} C_VEL
LIN {X 0,Y 319.854,Z 246.266,A -85,B 0,C 180,E1 -15292.424,E2 -15292.424} C_VEL
LIN {X 0,Y 319.735,Z 246.283,A -85,B 0,C 180,E1 -15294.956,E2 -15294.956} C_VEL
LIN {X 0,Y 319.99,Z 246.25,A -85,B 0,C 180,E1 -15297.482,E2 -15297.482} C_VEL
LIN {X 0,Y 320.096,Z 246.238,A -85,B 0,C 180,E1 -15300,E2 -15300} C_VEL
LIN {X 0,Y 319.986,Z 246.25,A -85,B 0,C 180,E1 -15302.518,E2 -15302.518} C_VEL
LIN {X 0,Y 319.92,Z 246.258,A -85,B 0,C 180,E1 -15306.664,E2 -15306.664} C_VEL
LIN {X 0,Y 319.754,Z 246.281,A -85,B 0,C 180,E1 -15310.127,E2 -15310.127} C_VEL
LIN {X 0,Y 319.732,Z 246.285,A -85,B 0,C 180,E1 -15314.724,E2 -15314.724} C_VEL
LIN {X 0,Y 319.69,Z 246.288,A -85,B 0,C 180,E1 -15319.038,E2 -15319.038} C_VEL
LIN {X 0,Y 319.561,Z 246.303,A -85,B 0,C 180,E1 -15323.32,E2 -15323.32} C_VEL
LIN {X 0,Y 319.635,Z 246.295,A -85,B 0,C 180,E1 -15326.088,E2 -15326.088} C_VEL
LIN {X 0,Y 319.581,Z 246.303,A -85,B 0,C 180,E1 -15328.935,E2 -15328.935} C_VEL
LIN {X 0,Y 319.532,Z 246.308,A -85,B 0,C 180,E1 -15331.862,E2 -15331.862} C_VEL
LIN {X 0,Y 319.581,Z 246.303,A -85,B 0,C 180,E1 -15335.543,E2 -15335.543} C_VEL
LIN {X 0,Y 319.528,Z 246.307,A -85,B 0,C 180,E1 -15339.662,E2 -15339.662} C_VEL
LIN {X 0,Y 319.521,Z 246.311,A -85,B 0,C 180,E1 -15343.46,E2 -15343.46} C_VEL
LIN {X 0,Y 319.559,Z 246.374,A -85,B 0,C 180,E1 -15347.017,E2 -15347.017} C_VEL
LIN {X 0,Y 319.841,Z 249.357,A -85,B 0,C 180,E1 -15350.415,E2 -15350.415} C_VEL
LIN {X 0,Y 319.75,Z 252.372,A -85,B 0,C 180,E1 -15353.598,E2 -15353.598} C_VEL
LIN {X 0,Y 319.504,Z 255.468,A -85,B 0,C 180,E1 -15356.707,E2 -15356.707} C_VEL
LIN {X 0,Y 319.228,Z 258.428,A -85,B 0,C 180,E1 -15359.578,E2 -15359.578} C_VEL
LIN {X 0,Y 318.992,Z 261.197,A -85,B 0,C 180,E1 -15362.182,E2 -15362.182} C_VEL
LIN {X 0,Y 320.07,Z 264.479,A -85,B 0,C 180,E1 -15362.398,E2 -15362.398} C_VEL
LIN {X 0,Y 324.853,Z 278.798,A -85,B 0,C 180,E1 -15363.44,E2 -15363.44} C_VEL
LIN {X 0,Y 328.364,Z 292.269,A -85,B 0,C 180,E1 -15364.575,E2 -15364.575} C_VEL
LIN {X 0,Y 330.573,Z 303.621,A -85,B 0,C 180,E1 -15365.663,E2 -15365.663} C_VEL
LIN {X 0,Y 330.637,Z 307.88,A -85,B 0,C 180,E1 -15366.065,E2 -15366.065} C_VEL
LIN {X 0,Y 329.127,Z 320.057,A -85,B 0,C 180,E1 -15367.25,E2 -15367.25} C_VEL
LIN {X 0,Y 327.358,Z 331.321,A -85,B 0,C 180,E1 -15368.594,E2 -15368.594} C_VEL
LIN {X 0,Y 325.63,Z 341.816,A -85,B 0,C 180,E1 -15370.128,E2 -15370.128} C_VEL
LIN {X 0,Y 323.752,Z 352.236,A -85,B 0,C 180,E1 -15371.981,E2 -15371.981} C_VEL
LIN {X 0,Y 322.012,Z 361.418,A -85,B 0,C 180,E1 -15373.987,E2 -15373.987} C_VEL
LIN {X 0,Y 320.806,Z 369.058,A -85,B 0,C 180,E1 -15376.056,E2 -15376.056} C_VEL
LIN {X 0,Y 319.736,Z 374.794,A -85,B 0,C 180,E1 -15377.947,E2 -15377.947} C_VEL
LIN {X 0,Y 319.012,Z 379.507,A -85,B 0,C 180,E1 -15379.849,E2 -15379.849} C_VEL
LIN {X 0,Y 318.341,Z 384.387,A -85,B 0,C 180,E1 -15382.388,E2 -15382.388} C_VEL
LIN {X 0,Y 317.98,Z 387.782,A -85,B 0,C 180,E1 -15384.928,E2 -15384.928} C_VEL
LIN {X 0,Y 317.785,Z 389.797,A -85,B 0,C 180,E1 -15387.465,E2 -15387.465} C_VEL
LIN {X 0,Y 317.721,Z 390.487,A -85,B 0,C 180,E1 -15390,E2 -15390} C_VEL
LIN {X 0,Y 317.784,Z 389.86,A -85,B 0,C 180,E1 -15392.535,E2 -15392.535} C_VEL
LIN {X 0,Y 317.978,Z 387.9,A -85,B 0,C 180,E1 -15395.072,E2 -15395.072} C_VEL
LIN {X 0,Y 318.34,Z 384.563,A -85,B 0,C 180,E1 -15397.612,E2 -15397.612} C_VEL
LIN {X 0,Y 318.98,Z 379.748,A -85,B 0,C 180,E1 -15400.152,E2 -15400.152} C_VEL
LIN {X 0,Y 319.689,Z 375.099,A -85,B 0,C 180,E1 -15402.055,E2 -15402.055} C_VEL
LIN {X 0,Y 320.964,Z 368.334,A -85,B 0,C 180,E1 -15404.261,E2 -15404.261} C_VEL
LIN {X 0,Y 322.066,Z 360.975,A -85,B 0,C 180,E1 -15406.229,E2 -15406.229} C_VEL
LIN {X 0,Y 323.638,Z 352.776,A -85,B 0,C 180,E1 -15408.026,E2 -15408.026} C_VEL
LIN {X 0,Y 325.515,Z 342.466,A -85,B 0,C 180,E1 -15409.88,E2 -15409.88} C_VEL
LIN {X 0,Y 327.524,Z 330.929,A -85,B 0,C 180,E1 -15411.56,E2 -15411.56} C_VEL
LIN {X 0,Y 329.367,Z 318.781,A -85,B 0,C 180,E1 -15412.991,E2 -15412.991} C_VEL
LIN {X 0,Y 330.878,Z 306.448,A -85,B 0,C 180,E1 -15414.162,E2 -15414.162} C_VEL
LIN {X 0,Y 329.141,Z 295.866,A -85,B 0,C 180,E1 -15415.202,E2 -15415.202} C_VEL
LIN {X 0,Y 325.995,Z 282.727,A -85,B 0,C 180,E1 -15416.351,E2 -15416.351} C_VEL
LIN {X 0,Y 321.611,Z 268.84,A -85,B 0,C 180,E1 -15417.414,E2 -15417.414} C_VEL
LIN {X 0,Y 319.075,Z 261.766,A -85,B 0,C 180,E1 -15417.892,E2 -15417.892} C_VEL
LIN {X 0,Y 318.983,Z 261.216,A -85,B 0,C 180,E1 -15417.918,E2 -15417.918} C_VEL
LIN {X 0,Y 319.237,Z 258.113,A -85,B 0,C 180,E1 -15420.842,E2 -15420.842} C_VEL
LIN {X 0,Y 319.511,Z 255.52,A -85,B 0,C 180,E1 -15423.361,E2 -15423.361} C_VEL
LIN {X 0,Y 319.746,Z 252.491,A -85,B 0,C 180,E1 -15426.403,E2 -15426.403} C_VEL
LIN {X 0,Y 319.849,Z 249.338,A -85,B 0,C 180,E1 -15429.731,E2 -15429.731} C_VEL
LIN {X 0,Y 319.56,Z 246.488,A -85,B 0,C 180,E1 -15432.983,E2 -15432.983} C_VEL
LIN {X 0,Y 319.554,Z 246.309,A -85,B 0,C 180,E1 -15437.016,E2 -15437.016} C_VEL
LIN {X 0,Y 319.547,Z 246.307,A -85,B 0,C 180,E1 -15440.371,E2 -15440.371} C_VEL
LIN {X 0,Y 319.582,Z 246.304,A -85,B 0,C 180,E1 -15444.457,E2 -15444.457} C_VEL
LIN {X 0,Y 319.559,Z 246.303,A -85,B 0,C 180,E1 -15446.912,E2 -15446.912} C_VEL
LIN {X 0,Y 318.848,Z 246.394,A -85,B 0,C 180,E1 -15447.965,E2 -15447.965} C_VEL
LIN {X 0,Y 316.013,Z 246.747,A -85,B 0,C 180,E1 -15449.679,E2 -15449.679} C_VEL
LIN {X 0,Y 313.641,Z 247.043,A -85,B 0,C 180,E1 -15451.068,E2 -15451.068} C_VEL
LIN {X 0,Y 312.624,Z 247.169,A -85,B 0,C 180,E1 -15452.142,E2 -15452.142} C_VEL
LIN {X 0,Y 312.539,Z 247.176,A -85,B 0,C 180,E1 -15452.506,E2 -15452.506} C_VEL
LIN {X 0,Y 312.587,Z 247.168,A -85,B 0,C 180,E1 -15454.711,E2 -15454.711} C_VEL
LIN {X 0,Y 312.54,Z 247.181,A -85,B 0,C 180,E1 -15458.913,E2 -15458.913} C_VEL
LIN {X 0,Y 312.641,Z 247.166,A -85,B 0,C 180,E1 -15461.656,E2 -15461.656} C_VEL
LIN {X 0,Y 312.697,Z 247.16,A -85,B 0,C 180,E1 -15465.686,E2 -15465.686} C_VEL
LIN {X 0,Y 312.688,Z 247.158,A -85,B 0,C 180,E1 -15469.641,E2 -15469.641} C_VEL
LIN {X 0,Y 312.895,Z 247.136,A -85,B 0,C 180,E1 -15473.552,E2 -15473.552} C_VEL
LIN {X 0,Y 312.934,Z 247.128,A -85,B 0,C 180,E1 -15477.425,E2 -15477.425} C_VEL
LIN {X 0,Y 312.991,Z 247.123,A -85,B 0,C 180,E1 -15481.287,E2 -15481.287} C_VEL
LIN {X 0,Y 312.705,Z 247.158,A -85,B 0,C 180,E1 -15485.158,E2 -15485.158} C_VEL
LIN {X 0,Y 312.799,Z 247.145,A -85,B 0,C 180,E1 -15487.747,E2 -15487.747} C_VEL
LIN {X 0,Y 312.666,Z 247.163,A -85,B 0,C 180,E1 -15491.671,E2 -15491.671} C_VEL
LIN {X 0,Y 312.671,Z 247.164,A -85,B 0,C 180,E1 -15494.865,E2 -15494.865} C_VEL
LIN {X 0,Y 312.593,Z 247.172,A -85,B 0,C 180,E1 -15499.215,E2 -15499.215} C_VEL
LIN {X 0,Y 312.524,Z 247.181,A -85,B 0,C 180,E1 -15502.779,E2 -15502.779} C_VEL
LIN {X 0,Y 312.531,Z 247.175,A -85,B 0,C 180,E1 -15505.908,E2 -15505.908} C_VEL
LIN {X 0,Y 312.497,Z 247.185,A -85,B 0,C 180,E1 -15509.655,E2 -15509.655} C_VEL
LIN {X 0,Y 312.521,Z 247.181,A -85,B 0,C 180,E1 -15513.689,E2 -15513.689} C_VEL
LIN {X 0,Y 312.527,Z 247.185,A -85,B 0,C 180,E1 -15517.385,E2 -15517.385} C_VEL
LIN {X 0,Y 312.563,Z 247.341,A -85,B 0,C 180,E1 -15520.91,E2 -15520.91} C_VEL
LIN {X 0,Y 313.067,Z 250.464,A -85,B 0,C 180,E1 -15524.1,E2 -15524.1} C_VEL
LIN {X 0,Y 313.627,Z 254.331,A -85,B 0,C 180,E1 -15527.758,E2 -15527.758} C_VEL
LIN {X 0,Y 313.813,Z 256.368,A -85,B 0,C 180,E1 -15529.592,E2 -15529.592} C_VEL
LIN {X 0,Y 313.653,Z 260.087,A -85,B 0,C 180,E1 -15532.772,E2 -15532.772} C_VEL
LIN {X 0,Y 313.138,Z 264.244,A -85,B 0,C 180,E1 -15536.142,E2 -15536.142} C_VEL
LIN {X 0,Y 312.761,Z 267.741,A -85,B 0,C 180,E1 -15538.88,E2 -15538.88} C_VEL
LIN {X 0,Y 312.368,Z 271.105,A -85,B 0,C 180,E1 -15541.46,E2 -15541.46} C_VEL
LIN {X 0,Y 313.251,Z 274.27,A -85,B 0,C 180,E1 -15541.647,E2 -15541.647} C_VEL
LIN {X 0,Y 317.442,Z 288.199,A -85,B 0,C 180,E1 -15542.626,E2 -15542.626} C_VEL
LIN {X 0,Y 320.411,Z 301.013,A -85,B 0,C 180,E1 -15543.665,E2 -15543.665} C_VEL
LIN {X 0,Y 322.392,Z 313.274,A -85,B 0,C 180,E1 -15544.796,E2 -15544.796} C_VEL
LIN {X 0,Y 323.312,Z 321.115,A -85,B 0,C 180,E1 -15545.606,E2 -15545.606} C_VEL
LIN {X 0,Y 321.677,Z 333.236,A -85,B 0,C 180,E1 -15546.842,E2 -15546.842} C_VEL
LIN {X 0,Y 319.624,Z 345.467,A -85,B 0,C 180,E1 -15548.389,E2 -15548.389} C_VEL
LIN {X 0,Y 317.8,Z 355.567,A -85,B 0,C 180,E1 -15549.954,E2 -15549.954} C_VEL
LIN {X 0,Y 315.954,Z 365.612,A -85,B 0,C 180,E1 -15551.855,E2 -15551.855} C_VEL
LIN {X 0,Y 314.491,Z 373.874,A -85,B 0,C 180,E1 -15553.756,E2 -15553.756} C_VEL
LIN {X 0,Y 313.104,Z 381.94,A -85,B 0,C 180,E1 -15556.037,E2 -15556.037} C_VEL
LIN {X 0,Y 311.931,Z 388.366,A -85,B 0,C 180,E1 -15558.3,E2 -15558.3} C_VEL
LIN {X 0,Y 311.217,Z 394.068,A -85,B 0,C 180,E1 -15560.905,E2 -15560.905} C_VEL
LIN {X 0,Y 310.814,Z 398.207,A -85,B 0,C 180,E1 -15563.508,E2 -15563.508} C_VEL
LIN {X 0,Y 310.679,Z 400.911,A -85,B 0,C 180,E1 -15566.109,E2 -15566.109} C_VEL
LIN {X 0,Y 310.61,Z 402.248,A -85,B 0,C 180,E1 -15568.703,E2 -15568.703} C_VEL
LIN {X 0,Y 310.61,Z 402.243,A -85,B 0,C 180,E1 -15571.296,E2 -15571.296} C_VEL
LIN {X 0,Y 310.677,Z 400.898,A -85,B 0,C 180,E1 -15573.891,E2 -15573.891} C_VEL
LIN {X 0,Y 310.814,Z 398.185,A -85,B 0,C 180,E1 -15576.492,E2 -15576.492} C_VEL
LIN {X 0,Y 311.196,Z 394.032,A -85,B 0,C 180,E1 -15579.096,E2 -15579.096} C_VEL
LIN {X 0,Y 311.929,Z 388.316,A -85,B 0,C 180,E1 -15581.699,E2 -15581.699} C_VEL
LIN {X 0,Y 313.096,Z 381.88,A -85,B 0,C 180,E1 -15583.963,E2 -15583.963} C_VEL
LIN {X 0,Y 314.403,Z 374.041,A -85,B 0,C 180,E1 -15586.183,E2 -15586.183} C_VEL
LIN {X 0,Y 315.943,Z 365.521,A -85,B 0,C 180,E1 -15588.145,E2 -15588.145} C_VEL
LIN {X 0,Y 317.812,Z 355.457,A -85,B 0,C 180,E1 -15590.045,E2 -15590.045} C_VEL
LIN {X 0,Y 319.799,Z 344.229,A -85,B 0,C 180,E1 -15591.768,E2 -15591.768} C_VEL
LIN {X 0,Y 321.959,Z 331.596,A -85,B 0,C 180,E1 -15593.311,E2 -15593.311} C_VEL
LIN {X 0,Y 323.238,Z 320.892,A -85,B 0,C 180,E1 -15594.4,E2 -15594.4} C_VEL
LIN {X 0,Y 321.666,Z 308.354,A -85,B 0,C 180,E1 -15595.658,E2 -15595.658} C_VEL
LIN {X 0,Y 319.528,Z 296.781,A -85,B 0,C 180,E1 -15596.673,E2 -15596.673} C_VEL
LIN {X 0,Y 315.781,Z 282.389,A -85,B 0,C 180,E1 -15597.781,E2 -15597.781} C_VEL
LIN {X 0,Y 312.375,Z 271.356,A -85,B 0,C 180,E1 -15598.501,E2 -15598.501} C_VEL
LIN {X 0,Y 312.375,Z 270.91,A -85,B 0,C 180,E1 -15598.664,E2 -15598.664} C_VEL
LIN {X 0,Y 312.753,Z 267.402,A -85,B 0,C 180,E1 -15601.36,E2 -15601.36} C_VEL
LIN {X 0,Y 313.158,Z 263.873,A -85,B 0,C 180,E1 -15604.129,E2 -15604.129} C_VEL
LIN {X 0,Y 313.648,Z 260.05,A -85,B 0,C 180,E1 -15607.229,E2 -15607.229} C_VEL
LIN {X 0,Y 313.809,Z 258.144,A -85,B 0,C 180,E1 -15608.835,E2 -15608.835} C_VEL
LIN {X 0,Y 313.799,Z 256.222,A -85,B 0,C 180,E1 -15610.504,E2 -15610.504} C_VEL
LIN {X 0,Y 313.301,Z 252.264,A -85,B 0,C 180,E1 -15614.125,E2 -15614.125} C_VEL
LIN {X 0,Y 312.759,Z 248.475,A -85,B 0,C 180,E1 -15617.863,E2 -15617.863} C_VEL
LIN {X 0,Y 312.531,Z 247.182,A -85,B 0,C 180,E1 -15619.297,E2 -15619.297} C_VEL
LIN {X 0,Y 312.526,Z 247.185,A -85,B 0,C 180,E1 -15622.615,E2 -15622.615} C_VEL
LIN {X 0,Y 312.52,Z 247.185,A -85,B 0,C 180,E1 -15626.311,E2 -15626.311} C_VEL
LIN {X 0,Y 312.497,Z 247.185,A -85,B 0,C 180,E1 -15630.345,E2 -15630.345} C_VEL
LIN {X 0,Y 312.531,Z 247.182,A -85,B 0,C 180,E1 -15634.092,E2 -15634.092} C_VEL
LIN {X 0,Y 312.564,Z 247.178,A -85,B 0,C 180,E1 -15637.527,E2 -15637.527} C_VEL
LIN {X 0,Y 312.59,Z 247.173,A -85,B 0,C 180,E1 -15641.653,E2 -15641.653} C_VEL
LIN {X 0,Y 312.687,Z 247.157,A -85,B 0,C 180,E1 -15645.686,E2 -15645.686} C_VEL
LIN {X 0,Y 312.687,Z 247.154,A -85,B 0,C 180,E1 -15649.641,E2 -15649.641} C_VEL
LIN {X 0,Y 312.798,Z 247.146,A -85,B 0,C 180,E1 -15652.253,E2 -15652.253} C_VEL
LIN {X 0,Y 312.703,Z 247.158,A -85,B 0,C 180,E1 -15654.842,E2 -15654.842} C_VEL
LIN {X 0,Y 312.99,Z 247.122,A -85,B 0,C 180,E1 -15658.713,E2 -15658.713} C_VEL
LIN {X 0,Y 312.984,Z 247.124,A -85,B 0,C 180,E1 -15661.287,E2 -15661.287} C_VEL
LIN {X 0,Y 312.711,Z 247.159,A -85,B 0,C 180,E1 -15665.158,E2 -15665.158} C_VEL
LIN {X 0,Y 312.855,Z 247.14,A -85,B 0,C 180,E1 -15667.746,E2 -15667.746} C_VEL
LIN {X 0,Y 312.671,Z 247.163,A -85,B 0,C 180,E1 -15671.671,E2 -15671.671} C_VEL
LIN {X 0,Y 312.702,Z 247.16,A -85,B 0,C 180,E1 -15674.888,E2 -15674.888} C_VEL
LIN {X 0,Y 312.631,Z 247.169,A -85,B 0,C 180,E1 -15679.236,E2 -15679.236} C_VEL
LIN {X 0,Y 312.527,Z 247.182,A -85,B 0,C 180,E1 -15682.781,E2 -15682.781} C_VEL
LIN {X 0,Y 312.604,Z 247.171,A -85,B 0,C 180,E1 -15685.936,E2 -15685.936} C_VEL
LIN {X 0,Y 312.539,Z 247.179,A -85,B 0,C 180,E1 -15689.651,E2 -15689.651} C_VEL
LIN {X 0,Y 312.52,Z 247.182,A -85,B 0,C 180,E1 -15693.689,E2 -15693.689} C_VEL
LIN {X 0,Y 312.515,Z 247.184,A -85,B 0,C 180,E1 -15697.387,E2 -15697.387} C_VEL
LIN {X 0,Y 312.441,Z 247.195,A -85,B 0,C 180,E1 -15700.717,E2 -15700.717} C_VEL
LIN {X 0,Y 312.452,Z 247.192,A -85,B 0,C 180,E1 -15704.21,E2 -15704.21} C_VEL
LIN {X 0,Y 312.46,Z 247.191,A -85,B 0,C 180,E1 -15706.035,E2 -15706.035} C_VEL
LIN {X 0,Y 312.628,Z 248.248,A -85,B 0,C 180,E1 -15707.89,E2 -15707.89} C_VEL
LIN {X 0,Y 312.798,Z 250.991,A -85,B 0,C 180,E1 -15711.016,E2 -15711.016} C_VEL
LIN {X 0,Y 312.69,Z 254.021,A -85,B 0,C 180,E1 -15714.241,E2 -15714.241} C_VEL
LIN {X 0,Y 312.39,Z 257.062,A -85,B 0,C 180,E1 -15717.32,E2 -15717.32} C_VEL
LIN {X 0,Y 311.961,Z 261.328,A -85,B 0,C 180,E1 -15721.505,E2 -15721.505} C_VEL
LIN {X 0,Y 313.002,Z 264.611,A -85,B 0,C 180,E1 -15721.718,E2 -15721.718} C_VEL
LIN {X 0,Y 317.481,Z 277.457,A -85,B 0,C 180,E1 -15722.698,E2 -15722.698} C_VEL
LIN {X 0,Y 321.09,Z 290.471,A -85,B 0,C 180,E1 -15723.82,E2 -15723.82} C_VEL
LIN {X 0,Y 323.604,Z 302.82,A -85,B 0,C 180,E1 -15725.021,E2 -15725.021} C_VEL
LIN {X 0,Y 324.214,Z 306.985,A -85,B 0,C 180,E1 -15725.46,E2 -15725.46} C_VEL
LIN {X 0,Y 322.73,Z 319.108,A -85,B 0,C 180,E1 -15726.643,E2 -15726.643} C_VEL
LIN {X 0,Y 320.75,Z 331.46,A -85,B 0,C 180,E1 -15728.131,E2 -15728.131} C_VEL
LIN {X 0,Y 318.942,Z 341.955,A -85,B 0,C 180,E1 -15729.693,E2 -15729.693} C_VEL
LIN {X 0,Y 316.989,Z 352.374,A -85,B 0,C 180,E1 -15731.583,E2 -15731.583} C_VEL
LIN {X 0,Y 315.082,Z 362.012,A -85,B 0,C 180,E1 -15733.747,E2 -15733.747} C_VEL
LIN {X 0,Y 313.899,Z 369.195,A -85,B 0,C 180,E1 -15735.742,E2 -15735.742} C_VEL
LIN {X 0,Y 312.769,Z 374.931,A -85,B 0,C 180,E1 -15737.674,E2 -15737.674} C_VEL
LIN {X 0,Y 311.998,Z 379.643,A -85,B 0,C 180,E1 -15739.618,E2 -15739.618} C_VEL
LIN {X 0,Y 311.277,Z 384.523,A -85,B 0,C 180,E1 -15742.214,E2 -15742.214} C_VEL
LIN {X 0,Y 310.9,Z 387.918,A -85,B 0,C 180,E1 -15744.812,E2 -15744.812} C_VEL
LIN {X 0,Y 310.711,Z 389.932,A -85,B 0,C 180,E1 -15747.407,E2 -15747.407} C_VEL
LIN {X 0,Y 310.634,Z 390.622,A -85,B 0,C 180,E1 -15750,E2 -15750} C_VEL
LIN {X 0,Y 310.71,Z 389.994,A -85,B 0,C 180,E1 -15752.593,E2 -15752.593} C_VEL
LIN {X 0,Y 310.898,Z 388.034,A -85,B 0,C 180,E1 -15755.188,E2 -15755.188} C_VEL
LIN {X 0,Y 311.107,Z 386.542,A -85,B 0,C 180,E1 -15756.486,E2 -15756.486} C_VEL
LIN {X 0,Y 311.601,Z 382.483,A -85,B 0,C 180,E1 -15759.084,E2 -15759.084} C_VEL
LIN {X 0,Y 312.454,Z 376.873,A -85,B 0,C 180,E1 -15761.68,E2 -15761.68} C_VEL
LIN {X 0,Y 313.656,Z 370.533,A -85,B 0,C 180,E1 -15763.938,E2 -15763.938} C_VEL
LIN {X 0,Y 314.825,Z 363.948,A -85,B 0,C 180,E1 -15765.852,E2 -15765.852} C_VEL
LIN {X 0,Y 316.021,Z 357.357,A -85,B 0,C 180,E1 -15767.471,E2 -15767.471} C_VEL
LIN {X 0,Y 317.878,Z 348.01,A -85,B 0,C 180,E1 -15769.368,E2 -15769.368} C_VEL
LIN {X 0,Y 319.741,Z 337.658,A -85,B 0,C 180,E1 -15771.096,E2 -15771.096} C_VEL
LIN {X 0,Y 321.663,Z 326.23,A -85,B 0,C 180,E1 -15772.649,E2 -15772.649} C_VEL
LIN {X 0,Y 323.489,Z 314.077,A -85,B 0,C 180,E1 -15773.983,E2 -15773.983} C_VEL
LIN {X 0,Y 324.289,Z 307.678,A -85,B 0,C 180,E1 -15774.579,E2 -15774.579} C_VEL
LIN {X 0,Y 322.59,Z 297.213,A -85,B 0,C 180,E1 -15775.657,E2 -15775.657} C_VEL
LIN {X 0,Y 319.419,Z 283.913,A -85,B 0,C 180,E1 -15776.875,E2 -15776.875} C_VEL
LIN {X 0,Y 315.164,Z 270.364,A -85,B 0,C 180,E1 -15777.968,E2 -15777.968} C_VEL
LIN {X 0,Y 312.088,Z 262.081,A -85,B 0,C 180,E1 -15778.567,E2 -15778.567} C_VEL
LIN {X 0,Y 311.976,Z 261.287,A -85,B 0,C 180,E1 -15778.652,E2 -15778.652} C_VEL
LIN {X 0,Y 312.393,Z 257.181,A -85,B 0,C 180,E1 -15782.68,E2 -15782.68} C_VEL
LIN {X 0,Y 312.702,Z 253.918,A -85,B 0,C 180,E1 -15785.991,E2 -15785.991} C_VEL
LIN {X 0,Y 312.791,Z 251.108,A -85,B 0,C 180,E1 -15788.986,E2 -15788.986} C_VEL
LIN {X 0,Y 312.627,Z 248.361,A -85,B 0,C 180,E1 -15792.11,E2 -15792.11} C_VEL
LIN {X 0,Y 312.448,Z 247.194,A -85,B 0,C 180,E1 -15794.211,E2 -15794.211} C_VEL
LIN {X 0,Y 312.457,Z 247.192,A -85,B 0,C 180,E1 -15797.925,E2 -15797.925} C_VEL
LIN {X 0,Y 312.486,Z 247.185,A -85,B 0,C 180,E1 -15801.922,E2 -15801.922} C_VEL
LIN {X 0,Y 312.533,Z 247.181,A -85,B 0,C 180,E1 -15804.22,E2 -15804.22} C_VEL
LIN {X 0,Y 312.506,Z 247.184,A -85,B 0,C 180,E1 -15807.334,E2 -15807.334} C_VEL
LIN {X 0,Y 312.547,Z 247.179,A -85,B 0,C 180,E1 -15811.279,E2 -15811.279} C_VEL
LIN {X 0,Y 312.539,Z 247.176,A -85,B 0,C 180,E1 -15812.506,E2 -15812.506} C_VEL
LIN {X 0,Y 311.858,Z 247.264,A -85,B 0,C 180,E1 -15813.581,E2 -15813.581} C_VEL
LIN {X 0,Y 308.974,Z 247.618,A -85,B 0,C 180,E1 -15815.33,E2 -15815.33} C_VEL
LIN {X 0,Y 306.553,Z 247.925,A -85,B 0,C 180,E1 -15816.749,E2 -15816.749} C_VEL
LIN {X 0,Y 305.542,Z 248.05,A -85,B 0,C 180,E1 -15817.848,E2 -15817.848} C_VEL
LIN {X 0,Y 305.475,Z 248.057,A -85,B 0,C 180,E1 -15818.221,E2 -15818.221} C_VEL
LIN {X 0,Y 305.592,Z 248.044,A -85,B 0,C 180,E1 -15821.218,E2 -15821.218} C_VEL
LIN {X 0,Y 305.652,Z 248.038,A -85,B 0,C 180,E1 -15825.349,E2 -15825.349} C_VEL
LIN {X 0,Y 305.627,Z 248.038,A -85,B 0,C 180,E1 -15829.399,E2 -15829.399} C_VEL
LIN {X 0,Y 305.774,Z 248.021,A -85,B 0,C 180,E1 -15832.073,E2 -15832.073} C_VEL
LIN {X 0,Y 305.682,Z 248.031,A -85,B 0,C 180,E1 -15834.723,E2 -15834.723} C_VEL
LIN {X 0,Y 305.943,Z 248.001,A -85,B 0,C 180,E1 -15838.684,E2 -15838.684} C_VEL
LIN {X 0,Y 305.958,Z 247.999,A -85,B 0,C 180,E1 -15841.316,E2 -15841.316} C_VEL
LIN {X 0,Y 305.673,Z 248.034,A -85,B 0,C 180,E1 -15845.277,E2 -15845.277} C_VEL
LIN {X 0,Y 305.749,Z 248.024,A -85,B 0,C 180,E1 -15847.927,E2 -15847.927} C_VEL
LIN {X 0,Y 305.601,Z 248.042,A -85,B 0,C 180,E1 -15851.945,E2 -15851.945} C_VEL
LIN {X 0,Y 305.613,Z 248.044,A -85,B 0,C 180,E1 -15855.015,E2 -15855.015} C_VEL
LIN {X 0,Y 305.549,Z 248.051,A -85,B 0,C 180,E1 -15859.429,E2 -15859.429} C_VEL
LIN {X 0,Y 305.488,Z 248.057,A -85,B 0,C 180,E1 -15863.039,E2 -15863.039} C_VEL
LIN {X 0,Y 305.471,Z 248.055,A -85,B 0,C 180,E1 -15866.197,E2 -15866.197} C_VEL
LIN {X 0,Y 305.45,Z 248.064,A -85,B 0,C 180,E1 -15869.034,E2 -15869.034} C_VEL
LIN {X 0,Y 305.438,Z 248.063,A -85,B 0,C 180,E1 -15871.953,E2 -15871.953} C_VEL
LIN {X 0,Y 305.464,Z 248.064,A -85,B 0,C 180,E1 -15875.113,E2 -15875.113} C_VEL
LIN {X 0,Y 305.451,Z 248.065,A -85,B 0,C 180,E1 -15878.528,E2 -15878.528} C_VEL
LIN {X 0,Y 305.512,Z 248.15,A -85,B 0,C 180,E1 -15880.361,E2 -15880.361} C_VEL
LIN {X 0,Y 305.979,Z 251.194,A -85,B 0,C 180,E1 -15883.556,E2 -15883.556} C_VEL
LIN {X 0,Y 306.525,Z 254.9,A -85,B 0,C 180,E1 -15887.197,E2 -15887.197} C_VEL
LIN {X 0,Y 306.78,Z 258.054,A -85,B 0,C 180,E1 -15890.1,E2 -15890.1} C_VEL
LIN {X 0,Y 306.727,Z 259.962,A -85,B 0,C 180,E1 -15891.782,E2 -15891.782} C_VEL
LIN {X 0,Y 306.248,Z 263.777,A -85,B 0,C 180,E1 -15894.99,E2 -15894.99} C_VEL
LIN {X 0,Y 305.761,Z 267.805,A -85,B 0,C 180,E1 -15898.261,E2 -15898.261} C_VEL
LIN {X 0,Y 305.383,Z 270.957,A -85,B 0,C 180,E1 -15900.739,E2 -15900.739} C_VEL
LIN {X 0,Y 306.329,Z 274.231,A -85,B 0,C 180,E1 -15900.949,E2 -15900.949} C_VEL
LIN {X 0,Y 310.197,Z 286.738,A -85,B 0,C 180,E1 -15901.865,E2 -15901.865} C_VEL
LIN {X 0,Y 313.477,Z 300.368,A -85,B 0,C 180,E1 -15903.001,E2 -15903.001} C_VEL
LIN {X 0,Y 315.55,Z 312.345,A -85,B 0,C 180,E1 -15904.14,E2 -15904.14} C_VEL
LIN {X 0,Y 316.689,Z 322.459,A -85,B 0,C 180,E1 -15905.217,E2 -15905.217} C_VEL
LIN {X 0,Y 314.923,Z 334.423,A -85,B 0,C 180,E1 -15906.49,E2 -15906.49} C_VEL
LIN {X 0,Y 312.807,Z 346.406,A -85,B 0,C 180,E1 -15908.067,E2 -15908.067} C_VEL
LIN {X 0,Y 310.765,Z 357.22,A -85,B 0,C 180,E1 -15909.825,E2 -15909.825} C_VEL
LIN {X 0,Y 308.868,Z 366.968,A -85,B 0,C 180,E1 -15911.768,E2 -15911.768} C_VEL
LIN {X 0,Y 307.272,Z 375.572,A -85,B 0,C 180,E1 -15913.87,E2 -15913.87} C_VEL
LIN {X 0,Y 306.008,Z 382.818,A -85,B 0,C 180,E1 -15916.045,E2 -15916.045} C_VEL
LIN {X 0,Y 304.935,Z 388.231,A -85,B 0,C 180,E1 -15918.028,E2 -15918.028} C_VEL
LIN {X 0,Y 304.174,Z 393.934,A -85,B 0,C 180,E1 -15920.692,E2 -15920.692} C_VEL
LIN {X 0,Y 303.726,Z 398.072,A -85,B 0,C 180,E1 -15923.356,E2 -15923.356} C_VEL
LIN {X 0,Y 303.577,Z 400.776,A -85,B 0,C 180,E1 -15926.017,E2 -15926.017} C_VEL
LIN {X 0,Y 303.58,Z 401.614,A -85,B 0,C 180,E1 -15927.346,E2 -15927.346} C_VEL
LIN {X 0,Y 303.545,Z 402.279,A -85,B 0,C 180,E1 -15930,E2 -15930} C_VEL
LIN {X 0,Y 303.579,Z 401.604,A -85,B 0,C 180,E1 -15932.654,E2 -15932.654} C_VEL
LIN {X 0,Y 303.617,Z 399.58,A -85,B 0,C 180,E1 -15935.313,E2 -15935.313} C_VEL
LIN {X 0,Y 303.919,Z 396.16,A -85,B 0,C 180,E1 -15937.975,E2 -15937.975} C_VEL
LIN {X 0,Y 304.518,Z 391.243,A -85,B 0,C 180,E1 -15940.64,E2 -15940.64} C_VEL
LIN {X 0,Y 305.273,Z 386.504,A -85,B 0,C 180,E1 -15942.633,E2 -15942.633} C_VEL
LIN {X 0,Y 306.531,Z 379.637,A -85,B 0,C 180,E1 -15944.947,E2 -15944.947} C_VEL
LIN {X 0,Y 308.061,Z 371.112,A -85,B 0,C 180,E1 -15947.252,E2 -15947.252} C_VEL
LIN {X 0,Y 309.736,Z 362.221,A -85,B 0,C 180,E1 -15949.209,E2 -15949.209} C_VEL
LIN {X 0,Y 311.776,Z 351.455,A -85,B 0,C 180,E1 -15951.141,E2 -15951.141} C_VEL
LIN {X 0,Y 313.838,Z 340.563,A -85,B 0,C 180,E1 -15952.724,E2 -15952.724} C_VEL
LIN {X 0,Y 315.905,Z 328.073,A -85,B 0,C 180,E1 -15954.198,E2 -15954.198} C_VEL
LIN {X 0,Y 316.629,Z 322.151,A -85,B 0,C 180,E1 -15954.798,E2 -15954.798} C_VEL
LIN {X 0,Y 314.985,Z 308.829,A -85,B 0,C 180,E1 -15956.194,E2 -15956.194} C_VEL
LIN {X 0,Y 312.707,Z 296.966,A -85,B 0,C 180,E1 -15957.279,E2 -15957.279} C_VEL
LIN {X 0,Y 309.169,Z 283.018,A -85,B 0,C 180,E1 -15958.395,E2 -15958.395} C_VEL
LIN {X 0,Y 305.456,Z 271.629,A -85,B 0,C 180,E1 -15959.195,E2 -15959.195} C_VEL
LIN {X 0,Y 305.378,Z 270.923,A -85,B 0,C 180,E1 -15959.261,E2 -15959.261} C_VEL
LIN {X 0,Y 305.988,Z 265.654,A -85,B 0,C 180,E1 -15963.452,E2 -15963.452} C_VEL
LIN {X 0,Y 306.501,Z 261.79,A -85,B 0,C 180,E1 -15966.626,E2 -15966.626} C_VEL
LIN {X 0,Y 306.812,Z 259.193,A -85,B 0,C 180,E1 -15968.847,E2 -15968.847} C_VEL
LIN {X 0,Y 306.627,Z 256.086,A -85,B 0,C 180,E1 -15971.659,E2 -15971.659} C_VEL
LIN {X 0,Y 306.12,Z 252.207,A -85,B 0,C 180,E1 -15975.374,E2 -15975.374} C_VEL
LIN {X 0,Y 305.757,Z 249.454,A -85,B 0,C 180,E1 -15978.196,E2 -15978.196} C_VEL
LIN {X 0,Y 305.479,Z 248.061,A -85,B 0,C 180,E1 -15979.896,E2 -15979.896} C_VEL
LIN {X 0,Y 305.482,Z 248.062,A -85,B 0,C 180,E1 -15983.632,E2 -15983.632} C_VEL
LIN {X 0,Y 305.465,Z 248.063,A -85,B 0,C 180,E1 -15986.483,E2 -15986.483} C_VEL
LIN {X 0,Y 305.431,Z 248.065,A -85,B 0,C 180,E1 -15989.588,E2 -15989.588} C_VEL
LIN {X 0,Y 305.458,Z 248.063,A -85,B 0,C 180,E1 -15992.603,E2 -15992.603} C_VEL
LIN {X 0,Y 305.475,Z 248.061,A -85,B 0,C 180,E1 -15995.536,E2 -15995.536} C_VEL
LIN {X 0,Y 305.501,Z 248.056,A -85,B 0,C 180,E1 -15999.814,E2 -15999.814} C_VEL
LIN {X 0,Y 305.548,Z 248.048,A -85,B 0,C 180,E1 -16002.601,E2 -16002.601} C_VEL
LIN {X 0,Y 305.628,Z 248.037,A -85,B 0,C 180,E1 -16005.348,E2 -16005.348} C_VEL
LIN {X 0,Y 305.625,Z 248.033,A -85,B 0,C 180,E1 -16009.399,E2 -16009.399} C_VEL
LIN {X 0,Y 305.748,Z 248.025,A -85,B 0,C 180,E1 -16012.073,E2 -16012.073} C_VEL
LIN {X 0,Y 305.672,Z 248.034,A -85,B 0,C 180,E1 -16014.723,E2 -16014.723} C_VEL
LIN {X 0,Y 305.957,Z 247.998,A -85,B 0,C 180,E1 -16018.684,E2 -16018.684} C_VEL
LIN {X 0,Y 305.952,Z 248.001,A -85,B 0,C 180,E1 -16021.316,E2 -16021.316} C_VEL
LIN {X 0,Y 305.843,Z 248.013,A -85,B 0,C 180,E1 -16026.598,E2 -16026.598} C_VEL
LIN {X 0,Y 305.705,Z 248.029,A -85,B 0,C 180,E1 -16029.261,E2 -16029.261} C_VEL
LIN {X 0,Y 305.591,Z 248.043,A -85,B 0,C 180,E1 -16033.296,E2 -16033.296} C_VEL
LIN {X 0,Y 305.595,Z 248.044,A -85,B 0,C 180,E1 -16036.02,E2 -16036.02} C_VEL
LIN {X 0,Y 305.577,Z 248.048,A -85,B 0,C 180,E1 -16039.445,E2 -16039.445} C_VEL
LIN {X 0,Y 305.487,Z 248.058,A -85,B 0,C 180,E1 -16043.039,E2 -16043.039} C_VEL
LIN {X 0,Y 305.548,Z 248.05,A -85,B 0,C 180,E1 -16046.227,E2 -16046.227} C_VEL
LIN {X 0,Y 305.49,Z 248.058,A -85,B 0,C 180,E1 -16049.048,E2 -16049.048} C_VEL
LIN {X 0,Y 305.443,Z 248.063,A -85,B 0,C 180,E1 -16051.952,E2 -16051.952} C_VEL
LIN {X 0,Y 305.463,Z 248.061,A -85,B 0,C 180,E1 -16055.113,E2 -16055.113} C_VEL
LIN {X 0,Y 305.434,Z 248.065,A -85,B 0,C 180,E1 -16058.525,E2 -16058.525} C_VEL
LIN {X 0,Y 305.437,Z 248.068,A -85,B 0,C 180,E1 -16062.582,E2 -16062.582} C_VEL
LIN {X 0,Y 305.422,Z 248.13,A -85,B 0,C 180,E1 -16066.344,E2 -16066.344} C_VEL
LIN {X 0,Y 305.79,Z 251.126,A -85,B 0,C 180,E1 -16069.945,E2 -16069.945} C_VEL
LIN {X 0,Y 305.698,Z 254.425,A -85,B 0,C 180,E1 -16073.577,E2 -16073.577} C_VEL
LIN {X 0,Y 305.438,Z 257.19,A -85,B 0,C 180,E1 -16076.48,E2 -16076.48} C_VEL
LIN {X 0,Y 305.028,Z 261.066,A -85,B 0,C 180,E1 -16080.382,E2 -16080.382} C_VEL
LIN {X 0,Y 304.993,Z 261.569,A -85,B 0,C 180,E1 -16080.803,E2 -16080.803} C_VEL
LIN {X 0,Y 305.884,Z 264.498,A -85,B 0,C 180,E1 -16080.989,E2 -16080.989} C_VEL
LIN {X 0,Y 310.355,Z 276.76,A -85,B 0,C 180,E1 -16081.973,E2 -16081.973} C_VEL
LIN {X 0,Y 314.114,Z 290.169,A -85,B 0,C 180,E1 -16083.16,E2 -16083.16} C_VEL
LIN {X 0,Y 316.68,Z 302.276,A -85,B 0,C 180,E1 -16084.374,E2 -16084.374} C_VEL
LIN {X 0,Y 317.614,Z 308.233,A -85,B 0,C 180,E1 -16085.025,E2 -16085.025} C_VEL
LIN {X 0,Y 316.045,Z 320.479,A -85,B 0,C 180,E1 -16086.27,E2 -16086.27} C_VEL
LIN {X 0,Y 313.955,Z 332.769,A -85,B 0,C 180,E1 -16087.805,E2 -16087.805} C_VEL
LIN {X 0,Y 311.936,Z 344.009,A -85,B 0,C 180,E1 -16089.56,E2 -16089.56} C_VEL
LIN {X 0,Y 309.921,Z 354.05,A -85,B 0,C 180,E1 -16091.49,E2 -16091.49} C_VEL
LIN {X 0,Y 308.151,Z 362.615,A -85,B 0,C 180,E1 -16093.5,E2 -16093.5} C_VEL
LIN {X 0,Y 307,Z 369.332,A -85,B 0,C 180,E1 -16095.415,E2 -16095.415} C_VEL
LIN {X 0,Y 305.79,Z 375.068,A -85,B 0,C 180,E1 -16097.389,E2 -16097.389} C_VEL
LIN {X 0,Y 304.999,Z 379.78,A -85,B 0,C 180,E1 -16099.377,E2 -16099.377} C_VEL
LIN {X 0,Y 304.24,Z 384.659,A -85,B 0,C 180,E1 -16102.033,E2 -16102.033} C_VEL
LIN {X 0,Y 303.824,Z 388.053,A -85,B 0,C 180,E1 -16104.691,E2 -16104.691} C_VEL
LIN {X 0,Y 303.638,Z 390.067,A -85,B 0,C 180,E1 -16107.347,E2 -16107.347} C_VEL
LIN {X 0,Y 303.55,Z 390.756,A -85,B 0,C 180,E1 -16110,E2 -16110} C_VEL
LIN {X 0,Y 303.638,Z 390.128,A -85,B 0,C 180,E1 -16112.653,E2 -16112.653} C_VEL
LIN {X 0,Y 303.825,Z 388.169,A -85,B 0,C 180,E1 -16115.309,E2 -16115.309} C_VEL
LIN {X 0,Y 304.239,Z 384.831,A -85,B 0,C 180,E1 -16117.967,E2 -16117.967} C_VEL
LIN {X 0,Y 304.973,Z 380.016,A -85,B 0,C 180,E1 -16120.624,E2 -16120.624} C_VEL
LIN {X 0,Y 306.075,Z 373.567,A -85,B 0,C 180,E1 -16123.275,E2 -16123.275} C_VEL
LIN {X 0,Y 307.63,Z 366.378,A -85,B 0,C 180,E1 -16125.571,E2 -16125.571} C_VEL
LIN {X 0,Y 308.66,Z 360.199,A -85,B 0,C 180,E1 -16127.218,E2 -16127.218} C_VEL
LIN {X 0,Y 310.476,Z 351.422,A -85,B 0,C 180,E1 -16129.161,E2 -16129.161} C_VEL
LIN {X 0,Y 312.536,Z 340.785,A -85,B 0,C 180,E1 -16131.088,E2 -16131.088} C_VEL
LIN {X 0,Y 314.534,Z 330.02,A -85,B 0,C 180,E1 -16132.671,E2 -16132.671} C_VEL
LIN {X 0,Y 316.419,Z 318.473,A -85,B 0,C 180,E1 -16134.059,E2 -16134.059} C_VEL
LIN {X 0,Y 317.628,Z 308.012,A -85,B 0,C 180,E1 -16135.11,E2 -16135.11} C_VEL
LIN {X 0,Y 315.307,Z 295.087,A -85,B 0,C 180,E1 -16136.474,E2 -16136.474} C_VEL
LIN {X 0,Y 311.854,Z 281.69,A -85,B 0,C 180,E1 -16137.724,E2 -16137.724} C_VEL
LIN {X 0,Y 307.411,Z 268.233,A -85,B 0,C 180,E1 -16138.832,E2 -16138.832} C_VEL
LIN {X 0,Y 305.079,Z 261.992,A -85,B 0,C 180,E1 -16139.293,E2 -16139.293} C_VEL
LIN {X 0,Y 305.012,Z 261.451,A -85,B 0,C 180,E1 -16139.355,E2 -16139.355} C_VEL
LIN {X 0,Y 305.44,Z 257.308,A -85,B 0,C 180,E1 -16143.52,E2 -16143.52} C_VEL
LIN {X 0,Y 305.707,Z 254.278,A -85,B 0,C 180,E1 -16146.707,E2 -16146.707} C_VEL
LIN {X 0,Y 305.786,Z 251.242,A -85,B 0,C 180,E1 -16150.056,E2 -16150.056} C_VEL
LIN {X 0,Y 305.435,Z 248.243,A -85,B 0,C 180,E1 -16153.654,E2 -16153.654} C_VEL
LIN {X 0,Y 305.438,Z 248.068,A -85,B 0,C 180,E1 -16157.418,E2 -16157.418} C_VEL
LIN {X 0,Y 305.462,Z 248.061,A -85,B 0,C 180,E1 -16161.595,E2 -16161.595} C_VEL
LIN {X 0,Y 305.464,Z 248.061,A -85,B 0,C 180,E1 -16164.887,E2 -16164.887} C_VEL
LIN {X 0,Y 305.452,Z 248.062,A -85,B 0,C 180,E1 -16168.356,E2 -16168.356} C_VEL
LIN {X 0,Y 305.516,Z 248.055,A -85,B 0,C 180,E1 -16171.113,E2 -16171.113} C_VEL
LIN {X 0,Y 305.573,Z 248.045,A -85,B 0,C 180,E1 -16174.088,E2 -16174.088} C_VEL
LIN {X 0,Y 305.475,Z 248.057,A -85,B 0,C 180,E1 -16178.221,E2 -16178.221} C_VEL
LIN {X 0,Y 304.849,Z 248.14,A -85,B 0,C 180,E1 -16179.322,E2 -16179.322} C_VEL
LIN {X 0,Y 302.03,Z 248.494,A -85,B 0,C 180,E1 -16181.116,E2 -16181.116} C_VEL
LIN {X 0,Y 299.633,Z 248.79,A -85,B 0,C 180,E1 -16182.571,E2 -16182.571} C_VEL
LIN {X 0,Y 298.627,Z 248.913,A -85,B 0,C 180,E1 -16183.698,E2 -16183.698} C_VEL
LIN {X 0,Y 298.559,Z 248.919,A -85,B 0,C 180,E1 -16184.079,E2 -16184.079} C_VEL
LIN {X 0,Y 298.553,Z 248.921,A -85,B 0,C 180,E1 -16187.768,E2 -16187.768} C_VEL
LIN {X 0,Y 298.72,Z 248.9,A -85,B 0,C 180,E1 -16191.885,E2 -16191.885} C_VEL
LIN {X 0,Y 298.653,Z 248.907,A -85,B 0,C 180,E1 -16194.599,E2 -16194.599} C_VEL
LIN {X 0,Y 298.911,Z 248.878,A -85,B 0,C 180,E1 -16198.653,E2 -16198.653} C_VEL
LIN {X 0,Y 298.925,Z 248.876,A -85,B 0,C 180,E1 -16201.347,E2 -16201.347} C_VEL
LIN {X 0,Y 298.641,Z 248.91,A -85,B 0,C 180,E1 -16205.401,E2 -16205.401} C_VEL
LIN {X 0,Y 298.71,Z 248.902,A -85,B 0,C 180,E1 -16208.82,E2 -16208.82} C_VEL
LIN {X 0,Y 298.548,Z 248.923,A -85,B 0,C 180,E1 -16213.615,E2 -16213.615} C_VEL
LIN {X 0,Y 298.492,Z 248.929,A -85,B 0,C 180,E1 -16216.412,E2 -16216.412} C_VEL
LIN {X 0,Y 298.489,Z 248.931,A -85,B 0,C 180,E1 -16219.641,E2 -16219.641} C_VEL
LIN {X 0,Y 298.422,Z 248.937,A -85,B 0,C 180,E1 -16223.601,E2 -16223.601} C_VEL
LIN {X 0,Y 298.409,Z 248.938,A -85,B 0,C 180,E1 -16226.582,E2 -16226.582} C_VEL
LIN {X 0,Y 298.395,Z 248.941,A -85,B 0,C 180,E1 -16229.644,E2 -16229.644} C_VEL
LIN {X 0,Y 298.394,Z 248.942,A -85,B 0,C 180,E1 -16232.8,E2 -16232.8} C_VEL
LIN {X 0,Y 298.448,Z 248.939,A -85,B 0,C 180,E1 -16236.807,E2 -16236.807} C_VEL
LIN {X 0,Y 298.453,Z 249.091,A -85,B 0,C 180,E1 -16239.918,E2 -16239.918} C_VEL
LIN {X 0,Y 298.952,Z 252.127,A -85,B 0,C 180,E1 -16243.216,E2 -16243.216} C_VEL
LIN {X 0,Y 299.521,Z 255.993,A -85,B 0,C 180,E1 -16247.12,E2 -16247.12} C_VEL
LIN {X 0,Y 299.702,Z 257.922,A -85,B 0,C 180,E1 -16248.959,E2 -16248.959} C_VEL
LIN {X 0,Y 299.783,Z 259.836,A -85,B 0,C 180,E1 -16250.729,E2 -16250.729} C_VEL
LIN {X 0,Y 299.352,Z 263.639,A -85,B 0,C 180,E1 -16254.06,E2 -16254.06} C_VEL
LIN {X 0,Y 298.749,Z 268.212,A -85,B 0,C 180,E1 -16257.875,E2 -16257.875} C_VEL
LIN {X 0,Y 298.43,Z 270.815,A -85,B 0,C 180,E1 -16259.994,E2 -16259.994} C_VEL
LIN {X 0,Y 299.457,Z 274.204,A -85,B 0,C 180,E1 -16260.219,E2 -16260.219} C_VEL
LIN {X 0,Y 303.47,Z 286.969,A -85,B 0,C 180,E1 -16261.202,E2 -16261.202} C_VEL
LIN {X 0,Y 306.541,Z 299.633,A -85,B 0,C 180,E1 -16262.296,E2 -16262.296} C_VEL
LIN {X 0,Y 308.799,Z 312.209,A -85,B 0,C 180,E1 -16263.531,E2 -16263.531} C_VEL
LIN {X 0,Y 310.015,Z 324.313,A -85,B 0,C 180,E1 -16264.871,E2 -16264.871} C_VEL
LIN {X 0,Y 308.183,Z 335.586,A -85,B 0,C 180,E1 -16266.122,E2 -16266.122} C_VEL
LIN {X 0,Y 306.002,Z 347.345,A -85,B 0,C 180,E1 -16267.731,E2 -16267.731} C_VEL
LIN {X 0,Y 304.073,Z 357.087,A -85,B 0,C 180,E1 -16269.361,E2 -16269.361} C_VEL
LIN {X 0,Y 302.091,Z 366.835,A -85,B 0,C 180,E1 -16271.344,E2 -16271.344} C_VEL
LIN {X 0,Y 300.487,Z 375.05,A -85,B 0,C 180,E1 -16273.386,E2 -16273.386} C_VEL
LIN {X 0,Y 299.061,Z 382.684,A -85,B 0,C 180,E1 -16275.714,E2 -16275.714} C_VEL
LIN {X 0,Y 297.956,Z 388.097,A -85,B 0,C 180,E1 -16277.743,E2 -16277.743} C_VEL
LIN {X 0,Y 297.116,Z 393.799,A -85,B 0,C 180,E1 -16280.469,E2 -16280.469} C_VEL
LIN {X 0,Y 296.65,Z 397.937,A -85,B 0,C 180,E1 -16283.197,E2 -16283.197} C_VEL
LIN {X 0,Y 296.48,Z 400.641,A -85,B 0,C 180,E1 -16285.922,E2 -16285.922} C_VEL
LIN {X 0,Y 296.451,Z 401.979,A -85,B 0,C 180,E1 -16288.641,E2 -16288.641} C_VEL
LIN {X 0,Y 296.451,Z 401.974,A -85,B 0,C 180,E1 -16291.358,E2 -16291.358} C_VEL
LIN {X 0,Y 296.477,Z 400.627,A -85,B 0,C 180,E1 -16294.078,E2 -16294.078} C_VEL
LIN {X 0,Y 296.65,Z 397.914,A -85,B 0,C 180,E1 -16296.803,E2 -16296.803} C_VEL
LIN {X 0,Y 297.106,Z 393.759,A -85,B 0,C 180,E1 -16299.531,E2 -16299.531} C_VEL
LIN {X 0,Y 297.954,Z 388.043,A -85,B 0,C 180,E1 -16302.256,E2 -16302.256} C_VEL
LIN {X 0,Y 299.184,Z 381.605,A -85,B 0,C 180,E1 -16304.627,E2 -16304.627} C_VEL
LIN {X 0,Y 300.475,Z 374.844,A -85,B 0,C 180,E1 -16306.65,E2 -16306.65} C_VEL
LIN {X 0,Y 302.082,Z 366.735,A -85,B 0,C 180,E1 -16308.657,E2 -16308.657} C_VEL
LIN {X 0,Y 304.05,Z 356.967,A -85,B 0,C 180,E1 -16310.64,E2 -16310.64} C_VEL
LIN {X 0,Y 306.201,Z 346.127,A -85,B 0,C 180,E1 -16312.432,E2 -16312.432} C_VEL
LIN {X 0,Y 308.413,Z 334.116,A -85,B 0,C 180,E1 -16314.037,E2 -16314.037} C_VEL
LIN {X 0,Y 310.015,Z 323.568,A -85,B 0,C 180,E1 -16315.188,E2 -16315.188} C_VEL
LIN {X 0,Y 308.529,Z 310.743,A -85,B 0,C 180,E1 -16316.6,E2 -16316.6} C_VEL
LIN {X 0,Y 306.109,Z 297.861,A -85,B 0,C 180,E1 -16317.844,E2 -16317.844} C_VEL
LIN {X 0,Y 302.66,Z 284.174,A -85,B 0,C 180,E1 -16318.997,E2 -16318.997} C_VEL
LIN {X 0,Y 298.504,Z 271.459,A -85,B 0,C 180,E1 -16319.943,E2 -16319.943} C_VEL
LIN {X 0,Y 298.426,Z 270.798,A -85,B 0,C 180,E1 -16319.991,E2 -16319.991} C_VEL
LIN {X 0,Y 299.104,Z 265.501,A -85,B 0,C 180,E1 -16324.328,E2 -16324.328} C_VEL
LIN {X 0,Y 299.581,Z 261.692,A -85,B 0,C 180,E1 -16327.586,E2 -16327.586} C_VEL
LIN {X 0,Y 299.772,Z 259.734,A -85,B 0,C 180,E1 -16329.316,E2 -16329.316} C_VEL
LIN {X 0,Y 299.671,Z 257.531,A -85,B 0,C 180,E1 -16331.368,E2 -16331.368} C_VEL
LIN {X 0,Y 299.174,Z 253.631,A -85,B 0,C 180,E1 -16335.191,E2 -16335.191} C_VEL
LIN {X 0,Y 298.664,Z 250.138,A -85,B 0,C 180,E1 -16338.852,E2 -16338.852} C_VEL
LIN {X 0,Y 298.416,Z 248.941,A -85,B 0,C 180,E1 -16340.296,E2 -16340.296} C_VEL
LIN {X 0,Y 298.419,Z 248.942,A -85,B 0,C 180,E1 -16343.93,E2 -16343.93} C_VEL
LIN {X 0,Y 298.389,Z 248.945,A -85,B 0,C 180,E1 -16347.986,E2 -16347.986} C_VEL
LIN {X 0,Y 298.414,Z 248.939,A -85,B 0,C 180,E1 -16351.899,E2 -16351.899} C_VEL
LIN {X 0,Y 298.44,Z 248.936,A -85,B 0,C 180,E1 -16354.92,E2 -16354.92} C_VEL
LIN {X 0,Y 298.418,Z 248.939,A -85,B 0,C 180,E1 -16357.864,E2 -16357.864} C_VEL
LIN {X 0,Y 298.509,Z 248.928,A -85,B 0,C 180,E1 -16360.755,E2 -16360.755} C_VEL
LIN {X 0,Y 298.587,Z 248.916,A -85,B 0,C 180,E1 -16364.994,E2 -16364.994} C_VEL
LIN {X 0,Y 298.584,Z 248.91,A -85,B 0,C 180,E1 -16369.146,E2 -16369.146} C_VEL
LIN {X 0,Y 298.699,Z 248.904,A -85,B 0,C 180,E1 -16371.884,E2 -16371.884} C_VEL
LIN {X 0,Y 298.64,Z 248.91,A -85,B 0,C 180,E1 -16374.599,E2 -16374.599} C_VEL
LIN {X 0,Y 298.923,Z 248.875,A -85,B 0,C 180,E1 -16378.653,E2 -16378.653} C_VEL
LIN {X 0,Y 298.919,Z 248.877,A -85,B 0,C 180,E1 -16381.347,E2 -16381.347} C_VEL
LIN {X 0,Y 298.788,Z 248.891,A -85,B 0,C 180,E1 -16386.754,E2 -16386.754} C_VEL
LIN {X 0,Y 298.637,Z 248.91,A -85,B 0,C 180,E1 -16389.482,E2 -16389.482} C_VEL
LIN {X 0,Y 298.554,Z 248.919,A -85,B 0,C 180,E1 -16393.615,E2 -16393.615} C_VEL
LIN {X 0,Y 298.55,Z 248.923,A -85,B 0,C 180,E1 -16396.409,E2 -16396.409} C_VEL
LIN {X 0,Y 298.512,Z 248.926,A -85,B 0,C 180,E1 -16399.654,E2 -16399.654} C_VEL
LIN {X 0,Y 298.43,Z 248.936,A -85,B 0,C 180,E1 -16403.6,E2 -16403.6} C_VEL
LIN {X 0,Y 298.49,Z 248.928,A -85,B 0,C 180,E1 -16406.574,E2 -16406.574} C_VEL
LIN {X 0,Y 298.418,Z 248.938,A -85,B 0,C 180,E1 -16409.641,E2 -16409.641} C_VEL
LIN {X 0,Y 298.396,Z 248.941,A -85,B 0,C 180,E1 -16412.8,E2 -16412.8} C_VEL
LIN {X 0,Y 298.429,Z 248.938,A -85,B 0,C 180,E1 -16416.803,E2 -16416.803} C_VEL
LIN {X 0,Y 298.374,Z 248.942,A -85,B 0,C 180,E1 -16419.492,E2 -16419.492} C_VEL
LIN {X 0,Y 298.4,Z 248.943,A -85,B 0,C 180,E1 -16423.103,E2 -16423.103} C_VEL
LIN {X 0,Y 298.355,Z 248.947,A -85,B 0,C 180,E1 -16425.035,E2 -16425.035} C_VEL
LIN {X 0,Y 298.491,Z 249.759,A -85,B 0,C 180,E1 -16426.937,E2 -16426.937} C_VEL
LIN {X 0,Y 298.693,Z 251.307,A -85,B 0,C 180,E1 -16428.845,E2 -16428.845} C_VEL
LIN {X 0,Y 298.782,Z 253.082,A -85,B 0,C 180,E1 -16430.917,E2 -16430.917} C_VEL
LIN {X 0,Y 298.618,Z 255.812,A -85,B 0,C 180,E1 -16433.958,E2 -16433.958} C_VEL
LIN {X 0,Y 298.315,Z 258.857,A -85,B 0,C 180,E1 -16437.19,E2 -16437.19} C_VEL
LIN {X 0,Y 298.028,Z 261.697,A -85,B 0,C 180,E1 -16440.051,E2 -16440.051} C_VEL
LIN {X 0,Y 299.039,Z 264.842,A -85,B 0,C 180,E1 -16440.265,E2 -16440.265} C_VEL
LIN {X 0,Y 303.777,Z 277.988,A -85,B 0,C 180,E1 -16441.366,E2 -16441.366} C_VEL
LIN {X 0,Y 307.225,Z 290.098,A -85,B 0,C 180,E1 -16442.492,E2 -16442.492} C_VEL
LIN {X 0,Y 309.781,Z 301.741,A -85,B 0,C 180,E1 -16443.698,E2 -16443.698} C_VEL
LIN {X 0,Y 311.038,Z 309.521,A -85,B 0,C 180,E1 -16444.576,E2 -16444.576} C_VEL
LIN {X 0,Y 309.382,Z 321.725,A -85,B 0,C 180,E1 -16445.865,E2 -16445.865} C_VEL
LIN {X 0,Y 307.195,Z 334.032,A -85,B 0,C 180,E1 -16447.468,E2 -16447.468} C_VEL
LIN {X 0,Y 305.261,Z 344.148,A -85,B 0,C 180,E1 -16449.093,E2 -16449.093} C_VEL
LIN {X 0,Y 303.185,Z 354.187,A -85,B 0,C 180,E1 -16451.063,E2 -16451.063} C_VEL
LIN {X 0,Y 301.221,Z 363.23,A -85,B 0,C 180,E1 -16453.246,E2 -16453.246} C_VEL
LIN {X 0,Y 299.898,Z 370.474,A -85,B 0,C 180,E1 -16455.409,E2 -16455.409} C_VEL
LIN {X 0,Y 298.54,Z 376.876,A -85,B 0,C 180,E1 -16457.768,E2 -16457.768} C_VEL
LIN {X 0,Y 297.555,Z 382.549,A -85,B 0,C 180,E1 -16460.483,E2 -16460.483} C_VEL
LIN {X 0,Y 296.963,Z 386.669,A -85,B 0,C 180,E1 -16463.204,E2 -16463.204} C_VEL
LIN {X 0,Y 296.658,Z 389.362,A -85,B 0,C 180,E1 -16465.925,E2 -16465.925} C_VEL
LIN {X 0,Y 296.477,Z 390.711,A -85,B 0,C 180,E1 -16468.642,E2 -16468.642} C_VEL
LIN {X 0,Y 296.477,Z 390.742,A -85,B 0,C 180,E1 -16471.358,E2 -16471.358} C_VEL
LIN {X 0,Y 296.657,Z 389.451,A -85,B 0,C 180,E1 -16474.076,E2 -16474.076} C_VEL
LIN {X 0,Y 296.964,Z 386.811,A -85,B 0,C 180,E1 -16476.796,E2 -16476.796} C_VEL
LIN {X 0,Y 297.544,Z 382.751,A -85,B 0,C 180,E1 -16479.517,E2 -16479.517} C_VEL
LIN {X 0,Y 298.476,Z 377.141,A -85,B 0,C 180,E1 -16482.235,E2 -16482.235} C_VEL
LIN {X 0,Y 299.835,Z 370.801,A -85,B 0,C 180,E1 -16484.595,E2 -16484.595} C_VEL
LIN {X 0,Y 300.895,Z 365.37,A -85,B 0,C 180,E1 -16486.277,E2 -16486.277} C_VEL
LIN {X 0,Y 302.441,Z 357.623,A -85,B 0,C 180,E1 -16488.283,E2 -16488.283} C_VEL
LIN {X 0,Y 304.495,Z 348.274,A -85,B 0,C 180,E1 -16490.256,E2 -16490.256} C_VEL
LIN {X 0,Y 306.508,Z 337.921,A -85,B 0,C 180,E1 -16492.053,E2 -16492.053} C_VEL
LIN {X 0,Y 308.623,Z 326.491,A -85,B 0,C 180,E1 -16493.663,E2 -16493.663} C_VEL
LIN {X 0,Y 310.529,Z 314.339,A -85,B 0,C 180,E1 -16495.051,E2 -16495.051} C_VEL
LIN {X 0,Y 311.085,Z 309.504,A -85,B 0,C 180,E1 -16495.537,E2 -16495.537} C_VEL
LIN {X 0,Y 309.109,Z 297.957,A -85,B 0,C 180,E1 -16496.825,E2 -16496.825} C_VEL
LIN {X 0,Y 305.764,Z 284.395,A -85,B 0,C 180,E1 -16498.167,E2 -16498.167} C_VEL
LIN {X 0,Y 301.587,Z 271.468,A -85,B 0,C 180,E1 -16499.311,E2 -16499.311} C_VEL
LIN {X 0,Y 298.094,Z 262.146,A -85,B 0,C 180,E1 -16500.048,E2 -16500.048} C_VEL
LIN {X 0,Y 298.039,Z 261.602,A -85,B 0,C 180,E1 -16500.098,E2 -16500.098} C_VEL
LIN {X 0,Y 298.509,Z 257.458,A -85,B 0,C 180,E1 -16504.406,E2 -16504.406} C_VEL
LIN {X 0,Y 298.692,Z 254.425,A -85,B 0,C 180,E1 -16507.717,E2 -16507.717} C_VEL
LIN {X 0,Y 298.759,Z 252.896,A -85,B 0,C 180,E1 -16509.431,E2 -16509.431} C_VEL
LIN {X 0,Y 298.688,Z 251.375,A -85,B 0,C 180,E1 -16511.211,E2 -16511.211} C_VEL
LIN {X 0,Y 298.488,Z 249.826,A -85,B 0,C 180,E1 -16513.121,E2 -16513.121} C_VEL
LIN {X 0,Y 298.356,Z 248.95,A -85,B 0,C 180,E1 -16515.035,E2 -16515.035} C_VEL
LIN {X 0,Y 298.373,Z 248.947,A -85,B 0,C 180,E1 -16516.915,E2 -16516.915} C_VEL
LIN {X 0,Y 298.386,Z 248.943,A -85,B 0,C 180,E1 -16521.011,E2 -16521.011} C_VEL
LIN {X 0,Y 298.407,Z 248.941,A -85,B 0,C 180,E1 -16523.928,E2 -16523.928} C_VEL
LIN {X 0,Y 298.397,Z 248.941,A -85,B 0,C 180,E1 -16527.2,E2 -16527.2} C_VEL
LIN {X 0,Y 298.43,Z 248.938,A -85,B 0,C 180,E1 -16530.616,E2 -16530.616} C_VEL
LIN {X 0,Y 298.485,Z 248.93,A -85,B 0,C 180,E1 -16533.475,E2 -16533.475} C_VEL
LIN {X 0,Y 298.433,Z 248.936,A -85,B 0,C 180,E1 -16536.699,E2 -16536.699} C_VEL
LIN {X 0,Y 298.541,Z 248.924,A -85,B 0,C 180,E1 -16540.757,E2 -16540.757} C_VEL
LIN {X 0,Y 298.559,Z 248.919,A -85,B 0,C 180,E1 -16544.079,E2 -16544.079} C_VEL
LIN {X 0,Y 297.916,Z 249.001,A -85,B 0,C 180,E1 -16545.205,E2 -16545.205} C_VEL
LIN {X 0,Y 295.04,Z 249.358,A -85,B 0,C 180,E1 -16547.037,E2 -16547.037} C_VEL
LIN {X 0,Y 292.611,Z 249.663,A -85,B 0,C 180,E1 -16548.525,E2 -16548.525} C_VEL
LIN {X 0,Y 291.611,Z 249.784,A -85,B 0,C 180,E1 -16549.677,E2 -16549.677} C_VEL
LIN {X 0,Y 291.553,Z 249.792,A -85,B 0,C 180,E1 -16550.068,E2 -16550.068} C_VEL
LIN {X 0,Y 291.726,Z 249.772,A -85,B 0,C 180,E1 -16553.081,E2 -16553.081} C_VEL
LIN {X 0,Y 291.786,Z 249.763,A -85,B 0,C 180,E1 -16557.239,E2 -16557.239} C_VEL
LIN {X 0,Y 291.862,Z 249.754,A -85,B 0,C 180,E1 -16560,E2 -16560} C_VEL
LIN {X 0,Y 291.789,Z 249.761,A -85,B 0,C 180,E1 -16562.761,E2 -16562.761} C_VEL
LIN {X 0,Y 291.69,Z 249.775,A -85,B 0,C 180,E1 -16566.919,E2 -16566.919} C_VEL
LIN {X 0,Y 291.571,Z 249.791,A -85,B 0,C 180,E1 -16569.714,E2 -16569.714} C_VEL
LIN {X 0,Y 291.518,Z 249.798,A -85,B 0,C 180,E1 -16573.95,E2 -16573.95} C_VEL
LIN {X 0,Y 291.446,Z 249.806,A -85,B 0,C 180,E1 -16576.82,E2 -16576.82} C_VEL
LIN {X 0,Y 291.426,Z 249.81,A -85,B 0,C 180,E1 -16579.86,E2 -16579.86} C_VEL
LIN {X 0,Y 291.362,Z 249.818,A -85,B 0,C 180,E1 -16584.209,E2 -16584.209} C_VEL
LIN {X 0,Y 291.355,Z 249.818,A -85,B 0,C 180,E1 -16587.278,E2 -16587.278} C_VEL
LIN {X 0,Y 291.32,Z 249.823,A -85,B 0,C 180,E1 -16590.439,E2 -16590.439} C_VEL
LIN {X 0,Y 291.345,Z 249.819,A -85,B 0,C 180,E1 -16593.698,E2 -16593.698} C_VEL
LIN {X 0,Y 291.378,Z 249.82,A -85,B 0,C 180,E1 -16597.254,E2 -16597.254} C_VEL
LIN {X 0,Y 291.385,Z 249.953,A -85,B 0,C 180,E1 -16599.363,E2 -16599.363} C_VEL
LIN {X 0,Y 291.825,Z 252.633,A -85,B 0,C 180,E1 -16602.401,E2 -16602.401} C_VEL
LIN {X 0,Y 292.364,Z 256.207,A -85,B 0,C 180,E1 -16606.15,E2 -16606.15} C_VEL
LIN {X 0,Y 292.681,Z 259.704,A -85,B 0,C 180,E1 -16609.583,E2 -16609.583} C_VEL
LIN {X 0,Y 292.565,Z 262.804,A -85,B 0,C 180,E1 -16612.441,E2 -16612.441} C_VEL
LIN {X 0,Y 291.932,Z 267.306,A -85,B 0,C 180,E1 -16616.378,E2 -16616.378} C_VEL
LIN {X 0,Y 291.501,Z 270.677,A -85,B 0,C 180,E1 -16619.206,E2 -16619.206} C_VEL
LIN {X 0,Y 292.524,Z 274.034,A -85,B 0,C 180,E1 -16619.437,E2 -16619.437} C_VEL
LIN {X 0,Y 297.153,Z 288.552,A -85,B 0,C 180,E1 -16620.621,E2 -16620.621} C_VEL
LIN {X 0,Y 300.392,Z 302.463,A -85,B 0,C 180,E1 -16621.895,E2 -16621.895} C_VEL
LIN {X 0,Y 302.566,Z 315.783,A -85,B 0,C 180,E1 -16623.296,E2 -16623.296} C_VEL
LIN {X 0,Y 303.36,Z 325.542,A -85,B 0,C 180,E1 -16624.438,E2 -16624.438} C_VEL
LIN {X 0,Y 301.472,Z 336.749,A -85,B 0,C 180,E1 -16625.74,E2 -16625.74} C_VEL
LIN {X 0,Y 299.207,Z 348.285,A -85,B 0,C 180,E1 -16627.379,E2 -16627.379} C_VEL
LIN {X 0,Y 297.031,Z 358.74,A -85,B 0,C 180,E1 -16629.212,E2 -16629.212} C_VEL
LIN {X 0,Y 295.007,Z 368.191,A -85,B 0,C 180,E1 -16631.239,E2 -16631.239} C_VEL
LIN {X 0,Y 293.292,Z 376.527,A -85,B 0,C 180,E1 -16633.436,E2 -16633.436} C_VEL
LIN {X 0,Y 292.103,Z 382.549,A -85,B 0,C 180,E1 -16635.367,E2 -16635.367} C_VEL
LIN {X 0,Y 290.993,Z 387.963,A -85,B 0,C 180,E1 -16637.445,E2 -16637.445} C_VEL
LIN {X 0,Y 290.082,Z 393.664,A -85,B 0,C 180,E1 -16640.236,E2 -16640.236} C_VEL
LIN {X 0,Y 289.575,Z 397.803,A -85,B 0,C 180,E1 -16643.03,E2 -16643.03} C_VEL
LIN {X 0,Y 289.388,Z 400.507,A -85,B 0,C 180,E1 -16645.822,E2 -16645.822} C_VEL
LIN {X 0,Y 289.374,Z 401.845,A -85,B 0,C 180,E1 -16648.608,E2 -16648.608} C_VEL
LIN {X 0,Y 289.374,Z 401.839,A -85,B 0,C 180,E1 -16651.392,E2 -16651.392} C_VEL
LIN {X 0,Y 289.383,Z 400.491,A -85,B 0,C 180,E1 -16654.178,E2 -16654.178} C_VEL
LIN {X 0,Y 289.575,Z 397.778,A -85,B 0,C 180,E1 -16656.97,E2 -16656.97} C_VEL
